LIN {X 0,Y 305.412,Z 307.44,A -85,B 0,C 180,E1 -15880.589,E2 -15880.589} C_VEL
LIN {X 0,Y 305.423,Z 307.439,A -85,B 0,C 180,E1 -15883.655,E2 -15883.655} C_VEL
LIN {X 0,Y 305.438,Z 307.44,A -85,B 0,C 180,E1 -15887.418,E2 -15887.418} C_VEL
LIN {X 0,Y 305.462,Z 307.437,A -85,B 0,C 180,E1 -15891.594,E2 -15891.594} C_VEL
LIN {X 0,Y 305.463,Z 307.435,A -85,B 0,C 180,E1 -15894.886,E2 -15894.886} C_VEL
LIN {X 0,Y 305.507,Z 307.555,A -85,B 0,C 180,E1 -15897.763,E2 -15897.763} C_VEL
LIN {X 0,Y 308.158,Z 320.105,A -85,B 0,C 180,E1 -15901.383,E2 -15901.383} C_VEL
LIN {X 0,Y 309.521,Z 328.593,A -85,B 0,C 180,E1 -15903.719,E2 -15903.719} C_VEL
LIN {X 0,Y 308.772,Z 334.974,A -85,B 0,C 180,E1 -15905.332,E2 -15905.332} C_VEL
LIN {X 0,Y 312.598,Z 362.726,A -85,B 0,C 180,E1 -15906.277,E2 -15906.277} C_VEL
LIN {X 0,Y 314.573,Z 379.937,A -85,B 0,C 180,E1 -15906.819,E2 -15906.819} C_VEL
LIN {X 0,Y 313.206,Z 444.59,A -85,B 0,C 180,E1 -15908.312,E2 -15908.312} C_VEL
LIN {X 0,Y 312.354,Z 458.417,A -85,B 0,C 180,E1 -15908.899,E2 -15908.899} C_VEL
LIN {X 0,Y 311.373,Z 470.835,A -85,B 0,C 180,E1 -15909.693,E2 -15909.693} C_VEL
LIN {X 0,Y 309.988,Z 483.522,A -85,B 0,C 180,E1 -15910.807,E2 -15910.807} C_VEL
LIN {X 0,Y 308.712,Z 494.84,A -85,B 0,C 180,E1 -15912.1,E2 -15912.1} C_VEL
LIN {X 0,Y 307.441,Z 505.618,A -85,B 0,C 180,E1 -15913.671,E2 -15913.671} C_VEL
LIN {X 0,Y 306.35,Z 515.028,A -85,B 0,C 180,E1 -15915.382,E2 -15915.382} C_VEL
LIN {X 0,Y 305.278,Z 523.823,A -85,B 0,C 180,E1 -15917.366,E2 -15917.366} C_VEL
LIN {X 0,Y 304.494,Z 530.826,A -85,B 0,C 180,E1 -15919.359,E2 -15919.359} C_VEL
LIN {X 0,Y 304.015,Z 536.433,A -85,B 0,C 180,E1 -15921.357,E2 -15921.357} C_VEL
LIN {X 0,Y 303.752,Z 540.824,A -85,B 0,C 180,E1 -15923.356,E2 -15923.356} C_VEL
LIN {X 0,Y 303.695,Z 543.143,A -85,B 0,C 180,E1 -15924.688,E2 -15924.688} C_VEL
LIN {X 0,Y 303.704,Z 545.022,A -85,B 0,C 180,E1 -15926.018,E2 -15926.018} C_VEL
LIN {X 0,Y 303.684,Z 546.422,A -85,B 0,C 180,E1 -15927.346,E2 -15927.346} C_VEL
LIN {X 0,Y 303.71,Z 547.415,A -85,B 0,C 180,E1 -15928.673,E2 -15928.673} C_VEL
LIN {X 0,Y 303.765,Z 548.015,A -85,B 0,C 180,E1 -15929.999,E2 -15929.999} C_VEL
LIN {X 0,Y 303.684,Z 548.212,A -85,B 0,C 180,E1 -15931.325,E2 -15931.325} C_VEL
LIN {X 0,Y 303.656,Z 547.975,A -85,B 0,C 180,E1 -15932.652,E2 -15932.652} C_VEL
LIN {X 0,Y 303.659,Z 547.346,A -85,B 0,C 180,E1 -15933.981,E2 -15933.981} C_VEL
LIN {X 0,Y 303.659,Z 546.063,A -85,B 0,C 180,E1 -15935.61,E2 -15935.61} C_VEL
LIN {X 0,Y 303.947,Z 543.046,A -85,B 0,C 180,E1 -15937.974,E2 -15937.974} C_VEL
LIN {X 0,Y 304.413,Z 539.432,A -85,B 0,C 180,E1 -15939.97,E2 -15939.97} C_VEL
LIN {X 0,Y 305.165,Z 534.729,A -85,B 0,C 180,E1 -15941.962,E2 -15941.962} C_VEL
LIN {X 0,Y 306.652,Z 527.682,A -85,B 0,C 180,E1 -15944.262,E2 -15944.262} C_VEL
LIN {X 0,Y 308.048,Z 520.393,A -85,B 0,C 180,E1 -15946.15,E2 -15946.15} C_VEL
LIN {X 0,Y 309.601,Z 512.33,A -85,B 0,C 180,E1 -15947.845,E2 -15947.845} C_VEL
LIN {X 0,Y 311.414,Z 502.899,A -85,B 0,C 180,E1 -15949.443,E2 -15949.443} C_VEL
LIN {X 0,Y 313.302,Z 492.462,A -85,B 0,C 180,E1 -15950.861,E2 -15950.861} C_VEL
LIN {X 0,Y 315.207,Z 480.88,A -85,B 0,C 180,E1 -15952.101,E2 -15952.101} C_VEL
LIN {X 0,Y 316.925,Z 468.596,A -85,B 0,C 180,E1 -15953.093,E2 -15953.093} C_VEL
LIN {X 0,Y 318.276,Z 455.706,A -85,B 0,C 180,E1 -15953.851,E2 -15953.851} C_VEL
LIN {X 0,Y 319.195,Z 443.251,A -85,B 0,C 180,E1 -15954.339,E2 -15954.339} C_VEL
LIN {X 0,Y 320.912,Z 380.563,A -85,B 0,C 180,E1 -15955.776,E2 -15955.776} C_VEL
LIN {X 0,Y 316.937,Z 356.478,A -85,B 0,C 180,E1 -15956.79,E2 -15956.79} C_VEL
LIN {X 0,Y 313.018,Z 337.758,A -85,B 0,C 180,E1 -15957.693,E2 -15957.693} C_VEL
LIN {X 0,Y 311.649,Z 334.114,A -85,B 0,C 180,E1 -15957.962,E2 -15957.962} C_VEL
LIN {X 0,Y 309.652,Z 324.511,A -85,B 0,C 180,E1 -15960.862,E2 -15960.862} C_VEL
LIN {X 0,Y 307.394,Z 314.899,A -85,B 0,C 180,E1 -15963.933,E2 -15963.933} C_VEL
LIN {X 0,Y 305.469,Z 307.44,A -85,B 0,C 180,E1 -15966.496,E2 -15966.496} C_VEL
LIN {X 0,Y 305.455,Z 307.437,A -85,B 0,C 180,E1 -15970.107,E2 -15970.107} C_VEL
LIN {X 0,Y 305.422,Z 307.44,A -85,B 0,C 180,E1 -15973.654,E2 -15973.654} C_VEL
LIN {X 0,Y 305.452,Z 307.436,A -85,B 0,C 180,E1 -15977.414,E2 -15977.414} C_VEL
LIN {X 0,Y 305.472,Z 307.43,A -85,B 0,C 180,E1 -15981.597,E2 -15981.597} C_VEL
LIN {X 0,Y 305.459,Z 307.429,A -85,B 0,C 180,E1 -15984.886,E2 -15984.886} C_VEL
LIN {X 0,Y 305.445,Z 307.43,A -85,B 0,C 180,E1 -15988.355,E2 -15988.355} C_VEL
LIN {X 0,Y 305.509,Z 307.423,A -85,B 0,C 180,E1 -15991.113,E2 -15991.113} C_VEL
LIN {X 0,Y 305.567,Z 307.42,A -85,B 0,C 180,E1 -15994.088,E2 -15994.088} C_VEL
LIN {X 0,Y 305.522,Z 307.427,A -85,B 0,C 180,E1 -15998.405,E2 -15998.405} C_VEL
LIN {X 0,Y 305.586,Z 307.42,A -85,B 0,C 180,E1 -16001.218,E2 -16001.218} C_VEL
LIN {X 0,Y 305.645,Z 307.412,A -85,B 0,C 180,E1 -16005.349,E2 -16005.349} C_VEL
LIN {X 0,Y 305.635,Z 307.413,A -85,B 0,C 180,E1 -16009.4,E2 -16009.4} C_VEL
LIN {X 0,Y 305.809,Z 307.383,A -85,B 0,C 180,E1 -16012.075,E2 -16012.075} C_VEL
LIN {X 0,Y 305.686,Z 307.408,A -85,B 0,C 180,E1 -16014.724,E2 -16014.724} C_VEL
LIN {X 0,Y 305.954,Z 307.375,A -85,B 0,C 180,E1 -16018.684,E2 -16018.684} C_VEL
LIN {X 0,Y 305.954,Z 307.369,A -85,B 0,C 180,E1 -16021.317,E2 -16021.317} C_VEL
LIN {X 0,Y 305.849,Z 307.384,A -85,B 0,C 180,E1 -16026.598,E2 -16026.598} C_VEL
LIN {X 0,Y 305.732,Z 307.394,A -85,B 0,C 180,E1 -16029.26,E2 -16029.26} C_VEL
LIN {X 0,Y 305.586,Z 307.413,A -85,B 0,C 180,E1 -16033.297,E2 -16033.297} C_VEL
LIN {X 0,Y 305.591,Z 307.417,A -85,B 0,C 180,E1 -16036.021,E2 -16036.021} C_VEL
LIN {X 0,Y 305.573,Z 307.422,A -85,B 0,C 180,E1 -16039.445,E2 -16039.445} C_VEL
LIN {X 0,Y 305.488,Z 307.432,A -85,B 0,C 180,E1 -16043.042,E2 -16043.042} C_VEL
LIN {X 0,Y 305.529,Z 307.424,A -85,B 0,C 180,E1 -16046.222,E2 -16046.222} C_VEL
LIN {X 0,Y 305.486,Z 307.427,A -85,B 0,C 180,E1 -16049.048,E2 -16049.048} C_VEL
LIN {X 0,Y 305.44,Z 307.43,A -85,B 0,C 180,E1 -16051.953,E2 -16051.953} C_VEL
LIN {X 0,Y 305.46,Z 307.43,A -85,B 0,C 180,E1 -16055.114,E2 -16055.114} C_VEL
LIN {X 0,Y 305.433,Z 307.431,A -85,B 0,C 180,E1 -16058.526,E2 -16058.526} C_VEL
LIN {X 0,Y 305.438,Z 307.438,A -85,B 0,C 180,E1 -16061.858,E2 -16061.858} C_VEL
LIN {X 0,Y 305.399,Z 307.441,A -85,B 0,C 180,E1 -16065.512,E2 -16065.512} C_VEL
LIN {X 0,Y 305.411,Z 307.441,A -85,B 0,C 180,E1 -16068.139,E2 -16068.139} C_VEL
LIN {X 0,Y 305.461,Z 307.635,A -85,B 0,C 180,E1 -16071.682,E2 -16071.682} C_VEL
LIN {X 0,Y 306.086,Z 309.918,A -85,B 0,C 180,E1 -16072.456,E2 -16072.456} C_VEL
LIN {X 0,Y 313.915,Z 325.345,A -85,B 0,C 180,E1 -16073.763,E2 -16073.763} C_VEL
LIN {X 0,Y 321.808,Z 343.043,A -85,B 0,C 180,E1 -16075.052,E2 -16075.052} C_VEL
LIN {X 0,Y 321.882,Z 347.906,A -85,B 0,C 180,E1 -16075.182,E2 -16075.182} C_VEL
LIN {X 0,Y 319.74,Z 416.224,A -85,B 0,C 180,E1 -16076.715,E2 -16076.715} C_VEL
LIN {X 0,Y 319.076,Z 429.194,A -85,B 0,C 180,E1 -16077.248,E2 -16077.248} C_VEL
LIN {X 0,Y 317.86,Z 442.361,A -85,B 0,C 180,E1 -16078.045,E2 -16078.045} C_VEL
LIN {X 0,Y 316.322,Z 454.752,A -85,B 0,C 180,E1 -16079.084,E2 -16079.084} C_VEL
LIN {X 0,Y 314.924,Z 465.141,A -85,B 0,C 180,E1 -16080.229,E2 -16080.229} C_VEL
LIN {X 0,Y 313.272,Z 475.048,A -85,B 0,C 180,E1 -16081.577,E2 -16081.577} C_VEL
LIN {X 0,Y 311.518,Z 484.552,A -85,B 0,C 180,E1 -16083.18,E2 -16083.18} C_VEL
LIN {X 0,Y 309.735,Z 493.368,A -85,B 0,C 180,E1 -16085.041,E2 -16085.041} C_VEL
LIN {X 0,Y 307.976,Z 501.365,A -85,B 0,C 180,E1 -16087.175,E2 -16087.175} C_VEL
LIN {X 0,Y 306.664,Z 507.305,A -85,B 0,C 180,E1 -16089.194,E2 -16089.194} C_VEL
LIN {X 0,Y 305.632,Z 511.949,A -85,B 0,C 180,E1 -16091.221,E2 -16091.221} C_VEL
LIN {X 0,Y 305.076,Z 514.383,A -85,B 0,C 180,E1 -16092.575,E2 -16092.575} C_VEL
LIN {X 0,Y 304.652,Z 516.358,A -85,B 0,C 180,E1 -16093.93,E2 -16093.93} C_VEL
LIN {X 0,Y 304.191,Z 518.541,A -85,B 0,C 180,E1 -16096.019,E2 -16096.019} C_VEL
LIN {X 0,Y 303.846,Z 519.689,A -85,B 0,C 180,E1 -16097.986,E2 -16097.986} C_VEL
LIN {X 0,Y 303.634,Z 519.884,A -85,B 0,C 180,E1 -16100.676,E2 -16100.676} C_VEL
LIN {X 0,Y 303.703,Z 519.354,A -85,B 0,C 180,E1 -16102.02,E2 -16102.02} C_VEL
LIN {X 0,Y 303.857,Z 517.831,A -85,B 0,C 180,E1 -16104.027,E2 -16104.027} C_VEL
LIN {X 0,Y 304.029,Z 514.328,A -85,B 0,C 180,E1 -16106.688,E2 -16106.688} C_VEL
LIN {X 0,Y 304.459,Z 510.533,A -85,B 0,C 180,E1 -16108.678,E2 -16108.678} C_VEL
LIN {X 0,Y 304.937,Z 505.635,A -85,B 0,C 180,E1 -16110.661,E2 -16110.661} C_VEL
LIN {X 0,Y 305.759,Z 499.464,A -85,B 0,C 180,E1 -16112.636,E2 -16112.636} C_VEL
LIN {X 0,Y 306.778,Z 491.775,A -85,B 0,C 180,E1 -16114.6,E2 -16114.6} C_VEL
LIN {X 0,Y 307.98,Z 482.158,A -85,B 0,C 180,E1 -16116.552,E2 -16116.552} C_VEL
LIN {X 0,Y 309.261,Z 472.211,A -85,B 0,C 180,E1 -16118.166,E2 -16118.166} C_VEL
LIN {X 0,Y 310.521,Z 460.956,A -85,B 0,C 180,E1 -16119.609,E2 -16119.609} C_VEL
LIN {X 0,Y 311.568,Z 449.946,A -85,B 0,C 180,E1 -16120.726,E2 -16120.726} C_VEL
LIN {X 0,Y 312.416,Z 437.754,A -85,B 0,C 180,E1 -16121.682,E2 -16121.682} C_VEL
LIN {X 0,Y 313.208,Z 424.771,A -85,B 0,C 180,E1 -16122.391,E2 -16122.391} C_VEL
LIN {X 0,Y 313.644,Z 410.959,A -85,B 0,C 180,E1 -16122.867,E2 -16122.867} C_VEL
LIN {X 0,Y 315.279,Z 336.381,A -85,B 0,C 180,E1 -16124.543,E2 -16124.543} C_VEL
LIN {X 0,Y 313.144,Z 328.581,A -85,B 0,C 180,E1 -16124.877,E2 -16124.877} C_VEL
LIN {X 0,Y 305.913,Z 308.922,A -85,B 0,C 180,E1 -16125.893,E2 -16125.893} C_VEL
LIN {X 0,Y 305.603,Z 307.419,A -85,B 0,C 180,E1 -16126.363,E2 -16126.363} C_VEL
LIN {X 0,Y 305.5,Z 307.429,A -85,B 0,C 180,E1 -16130.187,E2 -16130.187} C_VEL
LIN {X 0,Y 305.479,Z 307.43,A -85,B 0,C 180,E1 -16134.465,E2 -16134.465} C_VEL
LIN {X 0,Y 305.459,Z 307.433,A -85,B 0,C 180,E1 -16137.398,E2 -16137.398} C_VEL
LIN {X 0,Y 305.435,Z 307.436,A -85,B 0,C 180,E1 -16140.413,E2 -16140.413} C_VEL
LIN {X 0,Y 305.47,Z 307.431,A -85,B 0,C 180,E1 -16144.079,E2 -16144.079} C_VEL
LIN {X 0,Y 305.459,Z 307.435,A -85,B 0,C 180,E1 -16146.743,E2 -16146.743} C_VEL
LIN {X 0,Y 305.414,Z 307.437,A -85,B 0,C 180,E1 -16150.59,E2 -16150.59} C_VEL
LIN {X 0,Y 305.425,Z 307.439,A -85,B 0,C 180,E1 -16153.656,E2 -16153.656} C_VEL
LIN {X 0,Y 305.44,Z 307.435,A -85,B 0,C 180,E1 -16157.418,E2 -16157.418} C_VEL
LIN {X 0,Y 305.404,Z 307.436,A -85,B 0,C 180,E1 -16158.391,E2 -16158.391} C_VEL
LIN {X 0,Y 304.724,Z 307.528,A -85,B 0,C 180,E1 -16159.492,E2 -16159.492} C_VEL
LIN {X 0,Y 301.902,Z 307.879,A -85,B 0,C 180,E1 -16161.287,E2 -16161.287} C_VEL
LIN {X 0,Y 299.516,Z 308.174,A -85,B 0,C 180,E1 -16162.742,E2 -16162.742} C_VEL
LIN {X 0,Y 298.485,Z 308.3,A -85,B 0,C 180,E1 -16163.868,E2 -16163.868} C_VEL
LIN {X 0,Y 298.395,Z 308.308,A -85,B 0,C 180,E1 -16164.25,E2 -16164.25} C_VEL
LIN {X 0,Y 298.393,Z 308.314,A -85,B 0,C 180,E1 -16167.986,E2 -16167.986} C_VEL
LIN {X 0,Y 298.416,Z 308.311,A -85,B 0,C 180,E1 -16171.899,E2 -16171.899} C_VEL
LIN {X 0,Y 298.429,Z 308.3,A -85,B 0,C 180,E1 -16174.918,E2 -16174.918} C_VEL
LIN {X 0,Y 298.407,Z 308.315,A -85,B 0,C 180,E1 -16177.862,E2 -16177.862} C_VEL
LIN {X 0,Y 298.508,Z 308.298,A -85,B 0,C 180,E1 -16180.754,E2 -16180.754} C_VEL
LIN {X 0,Y 298.591,Z 308.28,A -85,B 0,C 180,E1 -16184.994,E2 -16184.994} C_VEL
LIN {X 0,Y 298.587,Z 308.288,A -85,B 0,C 180,E1 -16189.146,E2 -16189.146} C_VEL
LIN {X 0,Y 298.703,Z 308.277,A -85,B 0,C 180,E1 -16191.884,E2 -16191.884} C_VEL
LIN {X 0,Y 298.632,Z 308.276,A -85,B 0,C 180,E1 -16194.598,E2 -16194.598} C_VEL
LIN {X 0,Y 298.907,Z 308.25,A -85,B 0,C 180,E1 -16198.652,E2 -16198.652} C_VEL
LIN {X 0,Y 298.914,Z 308.248,A -85,B 0,C 180,E1 -16201.347,E2 -16201.347} C_VEL
LIN {X 0,Y 298.737,Z 308.267,A -85,B 0,C 180,E1 -16206.755,E2 -16206.755} C_VEL
LIN {X 0,Y 298.629,Z 308.282,A -85,B 0,C 180,E1 -16209.482,E2 -16209.482} C_VEL
LIN {X 0,Y 298.548,Z 308.292,A -85,B 0,C 180,E1 -16213.615,E2 -16213.615} C_VEL
LIN {X 0,Y 298.488,Z 308.305,A -85,B 0,C 180,E1 -16216.412,E2 -16216.412} C_VEL
LIN {X 0,Y 298.449,Z 308.306,A -85,B 0,C 180,E1 -16219.618,E2 -16219.618} C_VEL
LIN {X 0,Y 298.424,Z 308.309,A -85,B 0,C 180,E1 -16223.6,E2 -16223.6} C_VEL
LIN {X 0,Y 298.41,Z 308.314,A -85,B 0,C 180,E1 -16226.582,E2 -16226.582} C_VEL
LIN {X 0,Y 298.364,Z 308.318,A -85,B 0,C 180,E1 -16229.647,E2 -16229.647} C_VEL
LIN {X 0,Y 298.396,Z 308.317,A -85,B 0,C 180,E1 -16232.8,E2 -16232.8} C_VEL
LIN {X 0,Y 298.43,Z 308.312,A -85,B 0,C 180,E1 -16236.802,E2 -16236.802} C_VEL
LIN {X 0,Y 298.376,Z 308.318,A -85,B 0,C 180,E1 -16239.491,E2 -16239.491} C_VEL
LIN {X 0,Y 298.373,Z 308.32,A -85,B 0,C 180,E1 -16243.097,E2 -16243.097} C_VEL
LIN {X 0,Y 298.373,Z 308.317,A -85,B 0,C 180,E1 -16246.914,E2 -16246.914} C_VEL
LIN {X 0,Y 298.387,Z 308.316,A -85,B 0,C 180,E1 -16251.01,E2 -16251.01} C_VEL
LIN {X 0,Y 298.418,Z 308.314,A -85,B 0,C 180,E1 -16253.929,E2 -16253.929} C_VEL
LIN {X 0,Y 298.478,Z 308.417,A -85,B 0,C 180,E1 -16257.366,E2 -16257.366} C_VEL
LIN {X 0,Y 301.069,Z 320.78,A -85,B 0,C 180,E1 -16261.028,E2 -16261.028} C_VEL
LIN {X 0,Y 302.543,Z 329.288,A -85,B 0,C 180,E1 -16263.437,E2 -16263.437} C_VEL
LIN {X 0,Y 301.955,Z 334.637,A -85,B 0,C 180,E1 -16264.826,E2 -16264.826} C_VEL
LIN {X 0,Y 305.753,Z 362.062,A -85,B 0,C 180,E1 -16265.792,E2 -16265.792} C_VEL
LIN {X 0,Y 307.897,Z 380.351,A -85,B 0,C 180,E1 -16266.388,E2 -16266.388} C_VEL
LIN {X 0,Y 306.579,Z 443.282,A -85,B 0,C 180,E1 -16267.863,E2 -16267.863} C_VEL
LIN {X 0,Y 305.743,Z 456.666,A -85,B 0,C 180,E1 -16268.42,E2 -16268.42} C_VEL
LIN {X 0,Y 304.699,Z 469.491,A -85,B 0,C 180,E1 -16269.228,E2 -16269.228} C_VEL
LIN {X 0,Y 303.478,Z 480.858,A -85,B 0,C 180,E1 -16270.202,E2 -16270.202} C_VEL
LIN {X 0,Y 302.022,Z 492.589,A -85,B 0,C 180,E1 -16271.514,E2 -16271.514} C_VEL
LIN {X 0,Y 300.825,Z 503.17,A -85,B 0,C 180,E1 -16273.02,E2 -16273.02} C_VEL
LIN {X 0,Y 299.703,Z 512.814,A -85,B 0,C 180,E1 -16274.733,E2 -16274.733} C_VEL
LIN {X 0,Y 298.472,Z 521.816,A -85,B 0,C 180,E1 -16276.727,E2 -16276.727} C_VEL
LIN {X 0,Y 297.546,Z 529.18,A -85,B 0,C 180,E1 -16278.762,E2 -16278.762} C_VEL
LIN {X 0,Y 297.093,Z 534.164,A -85,B 0,C 180,E1 -16280.468,E2 -16280.468} C_VEL
LIN {X 0,Y 296.777,Z 538.998,A -85,B 0,C 180,E1 -16282.515,E2 -16282.515} C_VEL
LIN {X 0,Y 296.62,Z 542.689,A -85,B 0,C 180,E1 -16284.561,E2 -16284.561} C_VEL
LIN {X 0,Y 296.616,Z 544.593,A -85,B 0,C 180,E1 -16285.923,E2 -16285.923} C_VEL
LIN {X 0,Y 296.607,Z 546.027,A -85,B 0,C 180,E1 -16287.283,E2 -16287.283} C_VEL
LIN {X 0,Y 296.622,Z 547.038,A -85,B 0,C 180,E1 -16288.641,E2 -16288.641} C_VEL
LIN {X 0,Y 296.673,Z 547.656,A -85,B 0,C 180,E1 -16289.999,E2 -16289.999} C_VEL
LIN {X 0,Y 296.596,Z 547.877,A -85,B 0,C 180,E1 -16291.357,E2 -16291.357} C_VEL
LIN {X 0,Y 296.579,Z 547.673,A -85,B 0,C 180,E1 -16292.716,E2 -16292.716} C_VEL
LIN {X 0,Y 296.572,Z 547.061,A -85,B 0,C 180,E1 -16294.076,E2 -16294.076} C_VEL
LIN {X 0,Y 296.587,Z 545.932,A -85,B 0,C 180,E1 -16295.591,E2 -16295.591} C_VEL
LIN {X 0,Y 296.887,Z 542.837,A -85,B 0,C 180,E1 -16298.165,E2 -16298.165} C_VEL
LIN {X 0,Y 297.398,Z 539.265,A -85,B 0,C 180,E1 -16300.208,E2 -16300.208} C_VEL
LIN {X 0,Y 298.183,Z 534.607,A -85,B 0,C 180,E1 -16302.246,E2 -16302.246} C_VEL
LIN {X 0,Y 299.769,Z 527.608,A -85,B 0,C 180,E1 -16304.597,E2 -16304.597} C_VEL
LIN {X 0,Y 301.357,Z 519.808,A -85,B 0,C 180,E1 -16306.664,E2 -16306.664} C_VEL
LIN {X 0,Y 303.168,Z 510.646,A -85,B 0,C 180,E1 -16308.586,E2 -16308.586} C_VEL
LIN {X 0,Y 305.175,Z 500.933,A -85,B 0,C 180,E1 -16310.208,E2 -16310.208} C_VEL
LIN {X 0,Y 307.202,Z 490.161,A -85,B 0,C 180,E1 -16311.647,E2 -16311.647} C_VEL
LIN {X 0,Y 308.945,Z 479.683,A -85,B 0,C 180,E1 -16312.75,E2 -16312.75} C_VEL
LIN {X 0,Y 310.577,Z 468.216,A -85,B 0,C 180,E1 -16313.681,E2 -16313.681} C_VEL
LIN {X 0,Y 311.967,Z 455.318,A -85,B 0,C 180,E1 -16314.452,E2 -16314.452} C_VEL
LIN {X 0,Y 312.933,Z 442.835,A -85,B 0,C 180,E1 -16314.947,E2 -16314.947} C_VEL
LIN {X 0,Y 314.672,Z 381.223,A -85,B 0,C 180,E1 -16316.387,E2 -16316.387} C_VEL
LIN {X 0,Y 310.614,Z 356.75,A -85,B 0,C 180,E1 -16317.455,E2 -16317.455} C_VEL
LIN {X 0,Y 306.958,Z 339.936,A -85,B 0,C 180,E1 -16318.311,E2 -16318.311} C_VEL
LIN {X 0,Y 304.432,Z 333.652,A -85,B 0,C 180,E1 -16318.813,E2 -16318.813} C_VEL
LIN {X 0,Y 301.993,Z 322.401,A -85,B 0,C 180,E1 -16322.36,E2 -16322.36} C_VEL
LIN {X 0,Y 299.372,Z 311.813,A -85,B 0,C 180,E1 -16325.936,E2 -16325.936} C_VEL
LIN {X 0,Y 298.41,Z 308.314,A -85,B 0,C 180,E1 -16327.223,E2 -16327.223} C_VEL
LIN {X 0,Y 298.381,Z 308.314,A -85,B 0,C 180,E1 -16331.261,E2 -16331.261} C_VEL
LIN {X 0,Y 298.351,Z 308.322,A -85,B 0,C 180,E1 -16335.034,E2 -16335.034} C_VEL
LIN {X 0,Y 298.381,Z 308.313,A -85,B 0,C 180,E1 -16338.738,E2 -16338.738} C_VEL
LIN {X 0,Y 298.41,Z 308.308,A -85,B 0,C 180,E1 -16342.241,E2 -16342.241} C_VEL
LIN {X 0,Y 298.404,Z 308.307,A -85,B 0,C 180,E1 -16345.581,E2 -16345.581} C_VEL
LIN {X 0,Y 298.388,Z 308.309,A -85,B 0,C 180,E1 -16348.79,E2 -16348.79} C_VEL
LIN {X 0,Y 298.455,Z 308.299,A -85,B 0,C 180,E1 -16351.904,E2 -16351.904} C_VEL
LIN {X 0,Y 298.482,Z 308.298,A -85,B 0,C 180,E1 -16354.924,E2 -16354.924} C_VEL
LIN {X 0,Y 298.454,Z 308.298,A -85,B 0,C 180,E1 -16359.316,E2 -16359.316} C_VEL
LIN {X 0,Y 298.534,Z 308.298,A -85,B 0,C 180,E1 -16362.179,E2 -16362.179} C_VEL
LIN {X 0,Y 298.59,Z 308.291,A -85,B 0,C 180,E1 -16364.995,E2 -16364.995} C_VEL
LIN {X 0,Y 298.59,Z 308.291,A -85,B 0,C 180,E1 -16369.147,E2 -16369.147} C_VEL
LIN {X 0,Y 298.755,Z 308.262,A -85,B 0,C 180,E1 -16371.886,E2 -16371.886} C_VEL
LIN {X 0,Y 298.657,Z 308.284,A -85,B 0,C 180,E1 -16374.599,E2 -16374.599} C_VEL
LIN {X 0,Y 298.92,Z 308.251,A -85,B 0,C 180,E1 -16378.653,E2 -16378.653} C_VEL
LIN {X 0,Y 298.92,Z 308.245,A -85,B 0,C 180,E1 -16381.348,E2 -16381.348} C_VEL
LIN {X 0,Y 298.795,Z 308.264,A -85,B 0,C 180,E1 -16386.754,E2 -16386.754} C_VEL
LIN {X 0,Y 298.677,Z 308.273,A -85,B 0,C 180,E1 -16389.481,E2 -16389.481} C_VEL
LIN {X 0,Y 298.549,Z 308.289,A -85,B 0,C 180,E1 -16393.616,E2 -16393.616} C_VEL
LIN {X 0,Y 298.546,Z 308.295,A -85,B 0,C 180,E1 -16396.409,E2 -16396.409} C_VEL
LIN {X 0,Y 298.508,Z 308.301,A -85,B 0,C 180,E1 -16399.655,E2 -16399.655} C_VEL
LIN {X 0,Y 298.455,Z 308.308,A -85,B 0,C 180,E1 -16403.598,E2 -16403.598} C_VEL
LIN {X 0,Y 298.484,Z 308.302,A -85,B 0,C 180,E1 -16406.575,E2 -16406.575} C_VEL
LIN {X 0,Y 298.414,Z 308.31,A -85,B 0,C 180,E1 -16409.642,E2 -16409.642} C_VEL
LIN {X 0,Y 298.393,Z 308.308,A -85,B 0,C 180,E1 -16412.801,E2 -16412.801} C_VEL
LIN {X 0,Y 298.44,Z 308.308,A -85,B 0,C 180,E1 -16416.807,E2 -16416.807} C_VEL
LIN {X 0,Y 298.384,Z 308.312,A -85,B 0,C 180,E1 -16421.088,E2 -16421.088} C_VEL
LIN {X 0,Y 298.398,Z 308.313,A -85,B 0,C 180,E1 -16423.104,E2 -16423.104} C_VEL
LIN {X 0,Y 298.37,Z 308.321,A -85,B 0,C 180,E1 -16426.916,E2 -16426.916} C_VEL
LIN {X 0,Y 298.362,Z 308.328,A -85,B 0,C 180,E1 -16430.899,E2 -16430.899} C_VEL
LIN {X 0,Y 298.905,Z 310.268,A -85,B 0,C 180,E1 -16431.587,E2 -16431.587} C_VEL
LIN {X 0,Y 300.751,Z 313.796,A -85,B 0,C 180,E1 -16431.916,E2 -16431.916} C_VEL
LIN {X 0,Y 308.446,Z 328.838,A -85,B 0,C 180,E1 -16433.244,E2 -16433.244} C_VEL
LIN {X 0,Y 315.724,Z 345.313,A -85,B 0,C 180,E1 -16434.478,E2 -16434.478} C_VEL
LIN {X 0,Y 313.433,Z 417.477,A -85,B 0,C 180,E1 -16436.142,E2 -16436.142} C_VEL
LIN {X 0,Y 312.713,Z 430.572,A -85,B 0,C 180,E1 -16436.71,E2 -16436.71} C_VEL
LIN {X 0,Y 311.474,Z 443.2,A -85,B 0,C 180,E1 -16437.501,E2 -16437.501} C_VEL
LIN {X 0,Y 309.881,Z 455.439,A -85,B 0,C 180,E1 -16438.559,E2 -16438.559} C_VEL
LIN {X 0,Y 308.405,Z 465.76,A -85,B 0,C 180,E1 -16439.723,E2 -16439.723} C_VEL
LIN {X 0,Y 306.527,Z 476.414,A -85,B 0,C 180,E1 -16441.219,E2 -16441.219} C_VEL
LIN {X 0,Y 304.694,Z 485.937,A -85,B 0,C 180,E1 -16442.901,E2 -16442.901} C_VEL
LIN {X 0,Y 302.801,Z 494.732,A -85,B 0,C 180,E1 -16444.85,E2 -16444.85} C_VEL
LIN {X 0,Y 301.019,Z 502.377,A -85,B 0,C 180,E1 -16446.98,E2 -16446.98} C_VEL
LIN {X 0,Y 299.867,Z 507.273,A -85,B 0,C 180,E1 -16448.7,E2 -16448.7} C_VEL
LIN {X 0,Y 298.743,Z 511.997,A -85,B 0,C 180,E1 -16450.771,E2 -16450.771} C_VEL
LIN {X 0,Y 297.916,Z 515.569,A -85,B 0,C 180,E1 -16452.85,E2 -16452.85} C_VEL
LIN {X 0,Y 297.319,Z 518.097,A -85,B 0,C 180,E1 -16454.93,E2 -16454.93} C_VEL
LIN {X 0,Y 297.052,Z 519.26,A -85,B 0,C 180,E1 -16456.315,E2 -16456.315} C_VEL
LIN {X 0,Y 296.802,Z 519.974,A -85,B 0,C 180,E1 -16457.696,E2 -16457.696} C_VEL
LIN {X 0,Y 296.54,Z 520.234,A -85,B 0,C 180,E1 -16460.451,E2 -16460.451} C_VEL
LIN {X 0,Y 296.606,Z 519.766,A -85,B 0,C 180,E1 -16461.828,E2 -16461.828} C_VEL
LIN {X 0,Y 296.765,Z 518.102,A -85,B 0,C 180,E1 -16464.076,E2 -16464.076} C_VEL
LIN {X 0,Y 296.937,Z 514.87,A -85,B 0,C 180,E1 -16466.609,E2 -16466.609} C_VEL
LIN {X 0,Y 297.379,Z 511.144,A -85,B 0,C 180,E1 -16468.647,E2 -16468.647} C_VEL
LIN {X 0,Y 297.858,Z 506.322,A -85,B 0,C 180,E1 -16470.677,E2 -16470.677} C_VEL
LIN {X 0,Y 298.685,Z 500.235,A -85,B 0,C 180,E1 -16472.698,E2 -16472.698} C_VEL
LIN {X 0,Y 299.731,Z 492.678,A -85,B 0,C 180,E1 -16474.708,E2 -16474.708} C_VEL
LIN {X 0,Y 300.747,Z 484.954,A -85,B 0,C 180,E1 -16476.374,E2 -16476.374} C_VEL
LIN {X 0,Y 302.138,Z 474.455,A -85,B 0,C 180,E1 -16478.192,E2 -16478.192} C_VEL
LIN {X 0,Y 303.422,Z 463.775,A -85,B 0,C 180,E1 -16479.668,E2 -16479.668} C_VEL
LIN {X 0,Y 304.527,Z 453.401,A -85,B 0,C 180,E1 -16480.808,E2 -16480.808} C_VEL
LIN {X 0,Y 305.47,Z 440.987,A -85,B 0,C 180,E1 -16481.867,E2 -16481.867} C_VEL
LIN {X 0,Y 306.371,Z 427.838,A -85,B 0,C 180,E1 -16482.672,E2 -16482.672} C_VEL
LIN {X 0,Y 306.864,Z 414.521,A -85,B 0,C 180,E1 -16483.198,E2 -16483.198} C_VEL
LIN {X 0,Y 308.72,Z 337.899,A -85,B 0,C 180,E1 -16484.961,E2 -16484.961} C_VEL
LIN {X 0,Y 306.496,Z 330.201,A -85,B 0,C 180,E1 -16485.31,E2 -16485.31} C_VEL
LIN {X 0,Y 299.55,Z 311.529,A -85,B 0,C 180,E1 -16486.301,E2 -16486.301} C_VEL
LIN {X 0,Y 298.745,Z 309.24,A -85,B 0,C 180,E1 -16486.442,E2 -16486.442} C_VEL
LIN {X 0,Y 298.534,Z 308.3,A -85,B 0,C 180,E1 -16486.762,E2 -16486.762} C_VEL
LIN {X 0,Y 298.488,Z 308.302,A -85,B 0,C 180,E1 -16489.64,E2 -16489.64} C_VEL
LIN {X 0,Y 298.425,Z 308.307,A -85,B 0,C 180,E1 -16493.601,E2 -16493.601} C_VEL
LIN {X 0,Y 298.412,Z 308.31,A -85,B 0,C 180,E1 -16496.583,E2 -16496.583} C_VEL
LIN {X 0,Y 298.398,Z 308.312,A -85,B 0,C 180,E1 -16499.644,E2 -16499.644} C_VEL
LIN {X 0,Y 298.398,Z 308.316,A -85,B 0,C 180,E1 -16502.801,E2 -16502.801} C_VEL
LIN {X 0,Y 298.433,Z 308.311,A -85,B 0,C 180,E1 -16506.803,E2 -16506.803} C_VEL
LIN {X 0,Y 298.379,Z 308.315,A -85,B 0,C 180,E1 -16509.492,E2 -16509.492} C_VEL
LIN {X 0,Y 298.375,Z 308.317,A -85,B 0,C 180,E1 -16513.097,E2 -16513.097} C_VEL
LIN {X 0,Y 298.376,Z 308.314,A -85,B 0,C 180,E1 -16516.915,E2 -16516.915} C_VEL
LIN {X 0,Y 298.359,Z 308.318,A -85,B 0,C 180,E1 -16521.018,E2 -16521.018} C_VEL
LIN {X 0,Y 298.395,Z 308.308,A -85,B 0,C 180,E1 -16524.25,E2 -16524.25} C_VEL
LIN {X 0,Y 297.698,Z 308.397,A -85,B 0,C 180,E1 -16525.377,E2 -16525.377} C_VEL
LIN {X 0,Y 294.797,Z 308.759,A -85,B 0,C 180,E1 -16527.211,E2 -16527.211} C_VEL
LIN {X 0,Y 292.389,Z 309.062,A -85,B 0,C 180,E1 -16528.7,E2 -16528.7} C_VEL
LIN {X 0,Y 291.416,Z 309.185,A -85,B 0,C 180,E1 -16529.854,E2 -16529.854} C_VEL
LIN {X 0,Y 291.368,Z 309.189,A -85,B 0,C 180,E1 -16530.245,E2 -16530.245} C_VEL
LIN {X 0,Y 291.353,Z 309.182,A -85,B 0,C 180,E1 -16534.265,E2 -16534.265} C_VEL
LIN {X 0,Y 291.364,Z 309.187,A -85,B 0,C 180,E1 -16537.298,E2 -16537.298} C_VEL
LIN {X 0,Y 291.445,Z 309.18,A -85,B 0,C 180,E1 -16540.269,E2 -16540.269} C_VEL
LIN {X 0,Y 291.503,Z 309.162,A -85,B 0,C 180,E1 -16544.665,E2 -16544.665} C_VEL
LIN {X 0,Y 291.533,Z 309.167,A -85,B 0,C 180,E1 -16548.88,E2 -16548.88} C_VEL
LIN {X 0,Y 291.656,Z 309.153,A -85,B 0,C 180,E1 -16551.687,E2 -16551.687} C_VEL
LIN {X 0,Y 291.602,Z 309.152,A -85,B 0,C 180,E1 -16554.467,E2 -16554.467} C_VEL
LIN {X 0,Y 291.875,Z 309.126,A -85,B 0,C 180,E1 -16558.62,E2 -16558.62} C_VEL
LIN {X 0,Y 291.88,Z 309.124,A -85,B 0,C 180,E1 -16561.379,E2 -16561.379} C_VEL
LIN {X 0,Y 291.69,Z 309.143,A -85,B 0,C 180,E1 -16566.919,E2 -16566.919} C_VEL
LIN {X 0,Y 291.572,Z 309.161,A -85,B 0,C 180,E1 -16569.714,E2 -16569.714} C_VEL
LIN {X 0,Y 291.519,Z 309.168,A -85,B 0,C 180,E1 -16573.95,E2 -16573.95} C_VEL
LIN {X 0,Y 291.432,Z 309.183,A -85,B 0,C 180,E1 -16576.821,E2 -16576.821} C_VEL
LIN {X 0,Y 291.395,Z 309.185,A -85,B 0,C 180,E1 -16579.841,E2 -16579.841} C_VEL
LIN {X 0,Y 291.363,Z 309.19,A -85,B 0,C 180,E1 -16584.208,E2 -16584.208} C_VEL
LIN {X 0,Y 291.354,Z 309.192,A -85,B 0,C 180,E1 -16587.278,E2 -16587.278} C_VEL
LIN {X 0,Y 291.307,Z 309.198,A -85,B 0,C 180,E1 -16590.44,E2 -16590.44} C_VEL
LIN {X 0,Y 291.346,Z 309.192,A -85,B 0,C 180,E1 -16593.698,E2 -16593.698} C_VEL
LIN {X 0,Y 291.361,Z 309.194,A -85,B 0,C 180,E1 -16597.249,E2 -16597.249} C_VEL
LIN {X 0,Y 291.303,Z 309.198,A -85,B 0,C 180,E1 -16600.647,E2 -16600.647} C_VEL
LIN {X 0,Y 291.284,Z 309.199,A -85,B 0,C 180,E1 -16604.403,E2 -16604.403} C_VEL
LIN {X 0,Y 291.297,Z 309.197,A -85,B 0,C 180,E1 -16608.411,E2 -16608.411} C_VEL
LIN {X 0,Y 291.337,Z 309.196,A -85,B 0,C 180,E1 -16611.155,E2 -16611.155} C_VEL
LIN {X 0,Y 291.362,Z 309.192,A -85,B 0,C 180,E1 -16614.625,E2 -16614.625} C_VEL
LIN {X 0,Y 291.409,Z 309.396,A -85,B 0,C 180,E1 -16616.981,E2 -16616.981} C_VEL
LIN {X 0,Y 293.711,Z 320.009,A -85,B 0,C 180,E1 -16620.23,E2 -16620.23} C_VEL
LIN {X 0,Y 295.507,Z 329.966,A -85,B 0,C 180,E1 -16623.135,E2 -16623.135} C_VEL
LIN {X 0,Y 295.188,Z 334.296,A -85,B 0,C 180,E1 -16624.299,E2 -16624.299} C_VEL
LIN {X 0,Y 299.234,Z 363.733,A -85,B 0,C 180,E1 -16625.367,E2 -16625.367} C_VEL
LIN {X 0,Y 301.219,Z 381.077,A -85,B 0,C 180,E1 -16625.945,E2 -16625.945} C_VEL
LIN {X 0,Y 299.869,Z 443.076,A -85,B 0,C 180,E1 -16627.431,E2 -16627.431} C_VEL
LIN {X 0,Y 299,Z 456.417,A -85,B 0,C 180,E1 -16627.999,E2 -16627.999} C_VEL
LIN {X 0,Y 297.934,Z 469.226,A -85,B 0,C 180,E1 -16628.825,E2 -16628.825} C_VEL
LIN {X 0,Y 296.563,Z 481.373,A -85,B 0,C 180,E1 -16629.901,E2 -16629.901} C_VEL
LIN {X 0,Y 295.081,Z 492.952,A -85,B 0,C 180,E1 -16631.243,E2 -16631.243} C_VEL
LIN {X 0,Y 293.853,Z 503.412,A -85,B 0,C 180,E1 -16632.783,E2 -16632.783} C_VEL
LIN {X 0,Y 292.777,Z 512.293,A -85,B 0,C 180,E1 -16634.404,E2 -16634.404} C_VEL
LIN {X 0,Y 291.534,Z 521.168,A -85,B 0,C 180,E1 -16636.405,E2 -16636.405} C_VEL
LIN {X 0,Y 290.522,Z 528.584,A -85,B 0,C 180,E1 -16638.487,E2 -16638.487} C_VEL
LIN {X 0,Y 290.058,Z 533.621,A -85,B 0,C 180,E1 -16640.234,E2 -16640.234} C_VEL
LIN {X 0,Y 289.705,Z 538.499,A -85,B 0,C 180,E1 -16642.332,E2 -16642.332} C_VEL
LIN {X 0,Y 289.556,Z 542.235,A -85,B 0,C 180,E1 -16644.428,E2 -16644.428} C_VEL
LIN {X 0,Y 289.533,Z 544.159,A -85,B 0,C 180,E1 -16645.823,E2 -16645.823} C_VEL
LIN {X 0,Y 289.532,Z 545.632,A -85,B 0,C 180,E1 -16647.216,E2 -16647.216} C_VEL
LIN {X 0,Y 289.536,Z 546.662,A -85,B 0,C 180,E1 -16648.608,E2 -16648.608} C_VEL
LIN {X 0,Y 289.583,Z 547.298,A -85,B 0,C 180,E1 -16649.999,E2 -16649.999} C_VEL
LIN {X 0,Y 289.512,Z 547.537,A -85,B 0,C 180,E1 -16651.39,E2 -16651.39} C_VEL
LIN {X 0,Y 289.504,Z 547.37,A -85,B 0,C 180,E1 -16652.782,E2 -16652.782} C_VEL
LIN {X 0,Y 289.48,Z 545.856,A -85,B 0,C 180,E1 -16655.498,E2 -16655.498} C_VEL
LIN {X 0,Y 289.581,Z 544.422,A -85,B 0,C 180,E1 -16656.969,E2 -16656.969} C_VEL
LIN {X 0,Y 290.005,Z 541.546,A -85,B 0,C 180,E1 -16659.062,E2 -16659.062} C_VEL
LIN {X 0,Y 290.642,Z 537.659,A -85,B 0,C 180,E1 -16661.153,E2 -16661.153} C_VEL
LIN {X 0,Y 291.635,Z 532.667,A -85,B 0,C 180,E1 -16663.234,E2 -16663.234} C_VEL
LIN {X 0,Y 293.128,Z 526.421,A -85,B 0,C 180,E1 -16665.291,E2 -16665.291} C_VEL
LIN {X 0,Y 294.806,Z 518.627,A -85,B 0,C 180,E1 -16667.342,E2 -16667.342} C_VEL
LIN {X 0,Y 296.458,Z 510.742,A -85,B 0,C 180,E1 -16669.023,E2 -16669.023} C_VEL
LIN {X 0,Y 298.519,Z 501.116,A -85,B 0,C 180,E1 -16670.679,E2 -16670.679} C_VEL
LIN {X 0,Y 300.632,Z 490.452,A -85,B 0,C 180,E1 -16672.145,E2 -16672.145} C_VEL
LIN {X 0,Y 302.436,Z 480.149,A -85,B 0,C 180,E1 -16673.268,E2 -16673.268} C_VEL
LIN {X 0,Y 304.27,Z 467.844,A -85,B 0,C 180,E1 -16674.294,E2 -16674.294} C_VEL
LIN {X 0,Y 305.717,Z 454.932,A -85,B 0,C 180,E1 -16675.077,E2 -16675.077} C_VEL
LIN {X 0,Y 306.71,Z 442.421,A -85,B 0,C 180,E1 -16675.58,E2 -16675.58} C_VEL
LIN {X 0,Y 308.536,Z 382.541,A -85,B 0,C 180,E1 -16676.998,E2 -16676.998} C_VEL
LIN {X 0,Y 304.787,Z 359.56,A -85,B 0,C 180,E1 -16678.028,E2 -16678.028} C_VEL
LIN {X 0,Y 301.379,Z 343.152,A -85,B 0,C 180,E1 -16678.874,E2 -16678.874} C_VEL
LIN {X 0,Y 297.207,Z 333.325,A -85,B 0,C 180,E1 -16679.676,E2 -16679.676} C_VEL
LIN {X 0,Y 294.65,Z 321.968,A -85,B 0,C 180,E1 -16683.403,E2 -16683.403} C_VEL
LIN {X 0,Y 292.54,Z 313.464,A -85,B 0,C 180,E1 -16686.38,E2 -16686.38} C_VEL
LIN {X 0,Y 291.361,Z 309.193,A -85,B 0,C 180,E1 -16687.983,E2 -16687.983} C_VEL
LIN {X 0,Y 291.323,Z 309.193,A -85,B 0,C 180,E1 -16691.595,E2 -16691.595} C_VEL
LIN {X 0,Y 291.287,Z 309.2,A -85,B 0,C 180,E1 -16695.598,E2 -16695.598} C_VEL
LIN {X 0,Y 291.329,Z 309.19,A -85,B 0,C 180,E1 -16699.357,E2 -16699.357} C_VEL
LIN {X 0,Y 291.404,Z 309.184,A -85,B 0,C 180,E1 -16702.919,E2 -16702.919} C_VEL
LIN {X 0,Y 291.341,Z 309.19,A -85,B 0,C 180,E1 -16706.301,E2 -16706.301} C_VEL
LIN {X 0,Y 291.38,Z 309.187,A -85,B 0,C 180,E1 -16710.261,E2 -16710.261} C_VEL
LIN {X 0,Y 291.411,Z 309.184,A -85,B 0,C 180,E1 -16714.272,E2 -16714.272} C_VEL
LIN {X 0,Y 291.385,Z 309.187,A -85,B 0,C 180,E1 -16717.3,E2 -16717.3} C_VEL
LIN {X 0,Y 291.454,Z 309.171,A -85,B 0,C 180,E1 -16720.27,E2 -16720.27} C_VEL
LIN {X 0,Y 291.551,Z 309.163,A -85,B 0,C 180,E1 -16724.624,E2 -16724.624} C_VEL
LIN {X 0,Y 291.533,Z 309.167,A -85,B 0,C 180,E1 -16728.881,E2 -16728.881} C_VEL
LIN {X 0,Y 291.705,Z 309.14,A -85,B 0,C 180,E1 -16731.689,E2 -16731.689} C_VEL
LIN {X 0,Y 291.628,Z 309.159,A -85,B 0,C 180,E1 -16734.469,E2 -16734.469} C_VEL
LIN {X 0,Y 291.887,Z 309.126,A -85,B 0,C 180,E1 -16738.621,E2 -16738.621} C_VEL
LIN {X 0,Y 291.887,Z 309.121,A -85,B 0,C 180,E1 -16741.38,E2 -16741.38} C_VEL
LIN {X 0,Y 291.743,Z 309.144,A -85,B 0,C 180,E1 -16746.918,E2 -16746.918} C_VEL
LIN {X 0,Y 291.626,Z 309.152,A -85,B 0,C 180,E1 -16749.712,E2 -16749.712} C_VEL
LIN {X 0,Y 291.519,Z 309.166,A -85,B 0,C 180,E1 -16753.951,E2 -16753.951} C_VEL
LIN {X 0,Y 291.484,Z 309.172,A -85,B 0,C 180,E1 -16756.819,E2 -16756.819} C_VEL
LIN {X 0,Y 291.448,Z 309.179,A -85,B 0,C 180,E1 -16759.876,E2 -16759.876} C_VEL
LIN {X 0,Y 291.398,Z 309.185,A -85,B 0,C 180,E1 -16764.206,E2 -16764.206} C_VEL
LIN {X 0,Y 291.418,Z 309.186,A -85,B 0,C 180,E1 -16767.273,E2 -16767.273} C_VEL
LIN {X 0,Y 291.332,Z 309.194,A -85,B 0,C 180,E1 -16770.438,E2 -16770.438} C_VEL
LIN {X 0,Y 291.343,Z 309.193,A -85,B 0,C 180,E1 -16773.699,E2 -16773.699} C_VEL
LIN {X 0,Y 291.368,Z 309.189,A -85,B 0,C 180,E1 -16777.253,E2 -16777.253} C_VEL
LIN {X 0,Y 291.329,Z 309.192,A -85,B 0,C 180,E1 -16780.644,E2 -16780.644} C_VEL
LIN {X 0,Y 291.289,Z 309.201,A -85,B 0,C 180,E1 -16784.403,E2 -16784.403} C_VEL
LIN {X 0,Y 291.294,Z 309.201,A -85,B 0,C 180,E1 -16788.412,E2 -16788.412} C_VEL
LIN {X 0,Y 291.308,Z 309.308,A -85,B 0,C 180,E1 -16790.167,E2 -16790.167} C_VEL
LIN {X 0,Y 291.651,Z 310.648,A -85,B 0,C 180,E1 -16790.655,E2 -16790.655} C_VEL
LIN {X 0,Y 300.51,Z 327.304,A -85,B 0,C 180,E1 -16792.264,E2 -16792.264} C_VEL
LIN {X 0,Y 307.448,Z 342.352,A -85,B 0,C 180,E1 -16793.493,E2 -16793.493} C_VEL
LIN {X 0,Y 309.515,Z 347.181,A -85,B 0,C 180,E1 -16793.854,E2 -16793.854} C_VEL
LIN {X 0,Y 307.262,Z 417.17,A -85,B 0,C 180,E1 -16795.495,E2 -16795.495} C_VEL
LIN {X 0,Y 306.522,Z 430.337,A -85,B 0,C 180,E1 -16796.065,E2 -16796.065} C_VEL
LIN {X 0,Y 305.256,Z 442.887,A -85,B 0,C 180,E1 -16796.853,E2 -16796.853} C_VEL
LIN {X 0,Y 303.717,Z 454.508,A -85,B 0,C 180,E1 -16797.845,E2 -16797.845} C_VEL
LIN {X 0,Y 302.097,Z 465.059,A -85,B 0,C 180,E1 -16799.022,E2 -16799.022} C_VEL
LIN {X 0,Y 300.209,Z 475.899,A -85,B 0,C 180,E1 -16800.554,E2 -16800.554} C_VEL
LIN {X 0,Y 298.239,Z 485.605,A -85,B 0,C 180,E1 -16802.264,E2 -16802.264} C_VEL
LIN {X 0,Y 296.472,Z 493.444,A -85,B 0,C 180,E1 -16803.977,E2 -16803.977} C_VEL
LIN {X 0,Y 294.618,Z 501.14,A -85,B 0,C 180,E1 -16806.077,E2 -16806.077} C_VEL
LIN {X 0,Y 293.093,Z 507.249,A -85,B 0,C 180,E1 -16808.182,E2 -16808.182} C_VEL
LIN {X 0,Y 291.886,Z 512.048,A -85,B 0,C 180,E1 -16810.301,E2 -16810.301} C_VEL
LIN {X 0,Y 290.981,Z 515.692,A -85,B 0,C 180,E1 -16812.429,E2 -16812.429} C_VEL
LIN {X 0,Y 290.342,Z 518.286,A -85,B 0,C 180,E1 -16814.559,E2 -16814.559} C_VEL
LIN {X 0,Y 290.037,Z 519.493,A -85,B 0,C 180,E1 -16815.978,E2 -16815.978} C_VEL
LIN {X 0,Y 289.753,Z 520.261,A -85,B 0,C 180,E1 -16817.392,E2 -16817.392} C_VEL
LIN {X 0,Y 289.464,Z 520.583,A -85,B 0,C 180,E1 -16820.216,E2 -16820.216} C_VEL
LIN {X 0,Y 289.503,Z 520.162,A -85,B 0,C 180,E1 -16821.626,E2 -16821.626} C_VEL
LIN {X 0,Y 289.677,Z 518.381,A -85,B 0,C 180,E1 -16824.118,E2 -16824.118} C_VEL
LIN {X 0,Y 289.848,Z 515.41,A -85,B 0,C 180,E1 -16826.526,E2 -16826.526} C_VEL
LIN {X 0,Y 290.3,Z 511.754,A -85,B 0,C 180,E1 -16828.614,E2 -16828.614} C_VEL
LIN {X 0,Y 290.783,Z 507.007,A -85,B 0,C 180,E1 -16830.693,E2 -16830.693} C_VEL
LIN {X 0,Y 291.783,Z 499.892,A -85,B 0,C 180,E1 -16833.107,E2 -16833.107} C_VEL
LIN {X 0,Y 292.881,Z 492.128,A -85,B 0,C 180,E1 -16835.164,E2 -16835.164} C_VEL
LIN {X 0,Y 294.211,Z 482.444,A -85,B 0,C 180,E1 -16837.205,E2 -16837.205} C_VEL
LIN {X 0,Y 295.584,Z 472.393,A -85,B 0,C 180,E1 -16838.891,E2 -16838.891} C_VEL
LIN {X 0,Y 296.964,Z 461.013,A -85,B 0,C 180,E1 -16840.397,E2 -16840.397} C_VEL
LIN {X 0,Y 298.085,Z 449.861,A -85,B 0,C 180,E1 -16841.562,E2 -16841.562} C_VEL
LIN {X 0,Y 299.033,Z 437.334,A -85,B 0,C 180,E1 -16842.557,E2 -16842.557} C_VEL
LIN {X 0,Y 299.852,Z 423.888,A -85,B 0,C 180,E1 -16843.297,E2 -16843.297} C_VEL
LIN {X 0,Y 300.249,Z 411.4,A -85,B 0,C 180,E1 -16843.73,E2 -16843.73} C_VEL
LIN {X 0,Y 301.969,Z 338.21,A -85,B 0,C 180,E1 -16845.442,E2 -16845.442} C_VEL
LIN {X 0,Y 295.854,Z 320.471,A -85,B 0,C 180,E1 -16846.362,E2 -16846.362} C_VEL
LIN {X 0,Y 291.54,Z 309.57,A -85,B 0,C 180,E1 -16847.018,E2 -16847.018} C_VEL
LIN {X 0,Y 291.46,Z 309.181,A -85,B 0,C 180,E1 -16847.244,E2 -16847.244} C_VEL
LIN {X 0,Y 291.429,Z 309.182,A -85,B 0,C 180,E1 -16849.861,E2 -16849.861} C_VEL
LIN {X 0,Y 291.364,Z 309.186,A -85,B 0,C 180,E1 -16854.209,E2 -16854.209} C_VEL
LIN {X 0,Y 291.357,Z 309.19,A -85,B 0,C 180,E1 -16857.279,E2 -16857.279} C_VEL
LIN {X 0,Y 291.323,Z 309.194,A -85,B 0,C 180,E1 -16860.439,E2 -16860.439} C_VEL
LIN {X 0,Y 291.349,Z 309.191,A -85,B 0,C 180,E1 -16863.699,E2 -16863.699} C_VEL
LIN {X 0,Y 291.364,Z 309.193,A -85,B 0,C 180,E1 -16867.25,E2 -16867.25} C_VEL
LIN {X 0,Y 291.305,Z 309.195,A -85,B 0,C 180,E1 -16870.648,E2 -16870.648} C_VEL
LIN {X 0,Y 291.286,Z 309.198,A -85,B 0,C 180,E1 -16874.404,E2 -16874.404} C_VEL
LIN {X 0,Y 291.299,Z 309.192,A -85,B 0,C 180,E1 -16878.412,E2 -16878.412} C_VEL
LIN {X 0,Y 291.402,Z 309.184,A -85,B 0,C 180,E1 -16882.918,E2 -16882.918} C_VEL
LIN {X 0,Y 291.348,Z 309.186,A -85,B 0,C 180,E1 -16886.301,E2 -16886.301} C_VEL
LIN {X 0,Y 291.368,Z 309.189,A -85,B 0,C 180,E1 -16890.245,E2 -16890.245} C_VEL
LIN {X 0,Y 290.775,Z 309.265,A -85,B 0,C 180,E1 -16891.398,E2 -16891.398} C_VEL
LIN {X 0,Y 287.917,Z 309.621,A -85,B 0,C 180,E1 -16893.274,E2 -16893.274} C_VEL
LIN {X 0,Y 285.449,Z 309.927,A -85,B 0,C 180,E1 -16894.798,E2 -16894.798} C_VEL
LIN {X 0,Y 284.396,Z 310.056,A -85,B 0,C 180,E1 -16895.98,E2 -16895.98} C_VEL
LIN {X 0,Y 284.317,Z 310.064,A -85,B 0,C 180,E1 -16896.38,E2 -16896.38} C_VEL
LIN {X 0,Y 284.381,Z 310.063,A -85,B 0,C 180,E1 -16899.904,E2 -16899.904} C_VEL
LIN {X 0,Y 284.453,Z 310.04,A -85,B 0,C 180,E1 -16904.492,E2 -16904.492} C_VEL
LIN {X 0,Y 284.486,Z 310.046,A -85,B 0,C 180,E1 -16908.601,E2 -16908.601} C_VEL
LIN {X 0,Y 284.613,Z 310.029,A -85,B 0,C 180,E1 -16911.479,E2 -16911.479} C_VEL
LIN {X 0,Y 284.572,Z 310.027,A -85,B 0,C 180,E1 -16914.33,E2 -16914.33} C_VEL
LIN {X 0,Y 284.842,Z 310.002,A -85,B 0,C 180,E1 -16918.586,E2 -16918.586} C_VEL
LIN {X 0,Y 284.847,Z 310,A -85,B 0,C 180,E1 -16921.413,E2 -16921.413} C_VEL
LIN {X 0,Y 284.645,Z 310.019,A -85,B 0,C 180,E1 -16927.091,E2 -16927.091} C_VEL
LIN {X 0,Y 284.518,Z 310.041,A -85,B 0,C 180,E1 -16929.957,E2 -16929.957} C_VEL
LIN {X 0,Y 284.467,Z 310.049,A -85,B 0,C 180,E1 -16934.303,E2 -16934.303} C_VEL
LIN {X 0,Y 284.337,Z 310.067,A -85,B 0,C 180,E1 -16938.743,E2 -16938.743} C_VEL
LIN {X 0,Y 284.331,Z 310.066,A -85,B 0,C 180,E1 -16943.296,E2 -16943.296} C_VEL
LIN {X 0,Y 284.331,Z 310.068,A -85,B 0,C 180,E1 -16947.145,E2 -16947.145} C_VEL
LIN {X 0,Y 284.282,Z 310.074,A -85,B 0,C 180,E1 -16951.276,E2 -16951.276} C_VEL
LIN {X 0,Y 284.339,Z 310.068,A -85,B 0,C 180,E1 -16955.346,E2 -16955.346} C_VEL
LIN {X 0,Y 284.3,Z 310.07,A -85,B 0,C 180,E1 -16958.171,E2 -16958.171} C_VEL
LIN {X 0,Y 284.24,Z 310.077,A -85,B 0,C 180,E1 -16962.116,E2 -16962.116} C_VEL
LIN {X 0,Y 284.24,Z 310.076,A -85,B 0,C 180,E1 -16966.185,E2 -16966.185} C_VEL
LIN {X 0,Y 284.285,Z 310.072,A -85,B 0,C 180,E1 -16970.029,E2 -16970.029} C_VEL
LIN {X 0,Y 284.33,Z 310.071,A -85,B 0,C 180,E1 -16973.613,E2 -16973.613} C_VEL
LIN {X 0,Y 284.346,Z 310.223,A -85,B 0,C 180,E1 -16976.531,E2 -16976.531} C_VEL
LIN {X 0,Y 286.624,Z 320.737,A -85,B 0,C 180,E1 -16979.844,E2 -16979.844} C_VEL
LIN {X 0,Y 288.471,Z 330.639,A -85,B 0,C 180,E1 -16982.818,E2 -16982.818} C_VEL
LIN {X 0,Y 288.438,Z 333.938,A -85,B 0,C 180,E1 -16983.743,E2 -16983.743} C_VEL
LIN {X 0,Y 292.326,Z 362.357,A -85,B 0,C 180,E1 -16984.814,E2 -16984.814} C_VEL
LIN {X 0,Y 294.547,Z 382.324,A -85,B 0,C 180,E1 -16985.497,E2 -16985.497} C_VEL
LIN {X 0,Y 293.172,Z 442.822,A -85,B 0,C 180,E1 -16986.979,E2 -16986.979} C_VEL
LIN {X 0,Y 292.278,Z 456.137,A -85,B 0,C 180,E1 -16987.559,E2 -16987.559} C_VEL
LIN {X 0,Y 291.173,Z 468.933,A -85,B 0,C 180,E1 -16988.401,E2 -16988.401} C_VEL
LIN {X 0,Y 289.873,Z 480.273,A -85,B 0,C 180,E1 -16989.417,E2 -16989.417} C_VEL
LIN {X 0,Y 288.375,Z 491.999,A -85,B 0,C 180,E1 -16990.79,E2 -16990.79} C_VEL
LIN {X 0,Y 287,Z 502.556,A -85,B 0,C 180,E1 -16992.359,E2 -16992.359} C_VEL
LIN {X 0,Y 285.848,Z 511.752,A -85,B 0,C 180,E1 -16994.059,E2 -16994.059} C_VEL
LIN {X 0,Y 284.597,Z 520.51,A -85,B 0,C 180,E1 -16996.067,E2 -16996.067} C_VEL
LIN {X 0,Y 283.53,Z 527.986,A -85,B 0,C 180,E1 -16998.199,E2 -16998.199} C_VEL
LIN {X 0,Y 282.862,Z 534.868,A -85,B 0,C 180,E1 -17000.705,E2 -17000.705} C_VEL
LIN {X 0,Y 282.568,Z 539.396,A -85,B 0,C 180,E1 -17002.855,E2 -17002.855} C_VEL
LIN {X 0,Y 282.463,Z 541.962,A -85,B 0,C 180,E1 -17004.409,E2 -17004.409} C_VEL
LIN {X 0,Y 282.458,Z 545.234,A -85,B 0,C 180,E1 -17007.147,E2 -17007.147} C_VEL
LIN {X 0,Y 282.454,Z 546.285,A -85,B 0,C 180,E1 -17008.573,E2 -17008.573} C_VEL
LIN {X 0,Y 282.495,Z 546.94,A -85,B 0,C 180,E1 -17009.999,E2 -17009.999} C_VEL
LIN {X 0,Y 282.43,Z 547.198,A -85,B 0,C 180,E1 -17011.425,E2 -17011.425} C_VEL
LIN {X 0,Y 282.429,Z 547.063,A -85,B 0,C 180,E1 -17012.852,E2 -17012.852} C_VEL
LIN {X 0,Y 282.408,Z 545.723,A -85,B 0,C 180,E1 -17015.474,E2 -17015.474} C_VEL
LIN {X 0,Y 282.505,Z 544.176,A -85,B 0,C 180,E1 -17017.144,E2 -17017.144} C_VEL
LIN {X 0,Y 282.952,Z 541.342,A -85,B 0,C 180,E1 -17019.29,E2 -17019.29} C_VEL
LIN {X 0,Y 283.65,Z 537.498,A -85,B 0,C 180,E1 -17021.432,E2 -17021.432} C_VEL
LIN {X 0,Y 284.713,Z 532.552,A -85,B 0,C 180,E1 -17023.561,E2 -17023.561} C_VEL
LIN {X 0,Y 286.252,Z 526.357,A -85,B 0,C 180,E1 -17025.667,E2 -17025.667} C_VEL
LIN {X 0,Y 287.916,Z 519.15,A -85,B 0,C 180,E1 -17027.641,E2 -17027.641} C_VEL
LIN {X 0,Y 289.735,Z 510.839,A -85,B 0,C 180,E1 -17029.482,E2 -17029.482} C_VEL
LIN {X 0,Y 292.129,Z 500.231,A -85,B 0,C 180,E1 -17031.337,E2 -17031.337} C_VEL
LIN {X 0,Y 294.299,Z 489.452,A -85,B 0,C 180,E1 -17032.833,E2 -17032.833} C_VEL
LIN {X 0,Y 296.247,Z 478.956,A -85,B 0,C 180,E1 -17033.969,E2 -17033.969} C_VEL
LIN {X 0,Y 297.988,Z 467.474,A -85,B 0,C 180,E1 -17034.933,E2 -17034.933} C_VEL
LIN {X 0,Y 299.508,Z 454.545,A -85,B 0,C 180,E1 -17035.727,E2 -17035.727} C_VEL
LIN {X 0,Y 300.527,Z 442.005,A -85,B 0,C 180,E1 -17036.239,E2 -17036.239} C_VEL
LIN {X 0,Y 302.373,Z 383.406,A -85,B 0,C 180,E1 -17037.655,E2 -17037.655} C_VEL
LIN {X 0,Y 298.661,Z 360.312,A -85,B 0,C 180,E1 -17038.723,E2 -17038.723} C_VEL
LIN {X 0,Y 295.527,Z 345.542,A -85,B 0,C 180,E1 -17039.521,E2 -17039.521} C_VEL
LIN {X 0,Y 290.736,Z 335.022,A -85,B 0,C 180,E1 -17040.436,E2 -17040.436} C_VEL
LIN {X 0,Y 289.929,Z 332.84,A -85,B 0,C 180,E1 -17040.646,E2 -17040.646} C_VEL
LIN {X 0,Y 287.279,Z 321.088,A -85,B 0,C 180,E1 -17044.664,E2 -17044.664} C_VEL
LIN {X 0,Y 284.784,Z 311.84,A -85,B 0,C 180,E1 -17048.093,E2 -17048.093} C_VEL
LIN {X 0,Y 284.306,Z 310.07,A -85,B 0,C 180,E1 -17048.848,E2 -17048.848} C_VEL
LIN {X 0,Y 284.266,Z 310.074,A -85,B 0,C 180,E1 -17052.124,E2 -17052.124} C_VEL
LIN {X 0,Y 284.251,Z 310.074,A -85,B 0,C 180,E1 -17056.189,E2 -17056.189} C_VEL
LIN {X 0,Y 284.303,Z 310.068,A -85,B 0,C 180,E1 -17060.023,E2 -17060.023} C_VEL
LIN {X 0,Y 284.329,Z 310.066,A -85,B 0,C 180,E1 -17063.614,E2 -17063.614} C_VEL
LIN {X 0,Y 284.303,Z 310.067,A -85,B 0,C 180,E1 -17067.189,E2 -17067.189} C_VEL
LIN {X 0,Y 284.351,Z 310.063,A -85,B 0,C 180,E1 -17070.375,E2 -17070.375} C_VEL
LIN {X 0,Y 284.372,Z 310.059,A -85,B 0,C 180,E1 -17073.586,E2 -17073.586} C_VEL
LIN {X 0,Y 284.365,Z 310.057,A -85,B 0,C 180,E1 -17076.707,E2 -17076.707} C_VEL
LIN {X 0,Y 284.4,Z 310.059,A -85,B 0,C 180,E1 -17081.262,E2 -17081.262} C_VEL
LIN {X 0,Y 284.488,Z 310.041,A -85,B 0,C 180,E1 -17084.459,E2 -17084.459} C_VEL
LIN {X 0,Y 284.485,Z 310.042,A -85,B 0,C 180,E1 -17088.602,E2 -17088.602} C_VEL
LIN {X 0,Y 284.655,Z 310.019,A -85,B 0,C 180,E1 -17091.481,E2 -17091.481} C_VEL
LIN {X 0,Y 284.598,Z 310.034,A -85,B 0,C 180,E1 -17094.332,E2 -17094.332} C_VEL
LIN {X 0,Y 284.853,Z 310.002,A -85,B 0,C 180,E1 -17098.587,E2 -17098.587} C_VEL
LIN {X 0,Y 284.853,Z 309.997,A -85,B 0,C 180,E1 -17101.414,E2 -17101.414} C_VEL
LIN {X 0,Y 284.695,Z 310.023,A -85,B 0,C 180,E1 -17107.091,E2 -17107.091} C_VEL
LIN {X 0,Y 284.563,Z 310.033,A -85,B 0,C 180,E1 -17109.956,E2 -17109.956} C_VEL
LIN {X 0,Y 284.479,Z 310.043,A -85,B 0,C 180,E1 -17114.303,E2 -17114.303} C_VEL
LIN {X 0,Y 284.422,Z 310.049,A -85,B 0,C 180,E1 -17117.249,E2 -17117.249} C_VEL
LIN {X 0,Y 284.376,Z 310.06,A -85,B 0,C 180,E1 -17120.243,E2 -17120.243} C_VEL
LIN {X 0,Y 284.367,Z 310.061,A -85,B 0,C 180,E1 -17123.876,E2 -17123.876} C_VEL
LIN {X 0,Y 284.393,Z 310.062,A -85,B 0,C 180,E1 -17127.174,E2 -17127.174} C_VEL
LIN {X 0,Y 284.292,Z 310.069,A -85,B 0,C 180,E1 -17131.275,E2 -17131.275} C_VEL
LIN {X 0,Y 284.339,Z 310.06,A -85,B 0,C 180,E1 -17135.349,E2 -17135.349} C_VEL
LIN {X 0,Y 284.304,Z 310.063,A -85,B 0,C 180,E1 -17138.171,E2 -17138.171} C_VEL
LIN {X 0,Y 284.267,Z 310.075,A -85,B 0,C 180,E1 -17142.125,E2 -17142.125} C_VEL
LIN {X 0,Y 284.237,Z 310.078,A -85,B 0,C 180,E1 -17146.187,E2 -17146.187} C_VEL
LIN {X 0,Y 284.253,Z 310.113,A -85,B 0,C 180,E1 -17149.332,E2 -17149.332} C_VEL
LIN {X 0,Y 284.511,Z 311.244,A -85,B 0,C 180,E1 -17149.686,E2 -17149.686} C_VEL
LIN {X 0,Y 286.442,Z 314.675,A -85,B 0,C 180,E1 -17150.062,E2 -17150.062} C_VEL
LIN {X 0,Y 294.893,Z 330.409,A -85,B 0,C 180,E1 -17151.651,E2 -17151.651} C_VEL
LIN {X 0,Y 301.817,Z 345.461,A -85,B 0,C 180,E1 -17152.924,E2 -17152.924} C_VEL
LIN {X 0,Y 303.435,Z 349.255,A -85,B 0,C 180,E1 -17153.218,E2 -17153.218} C_VEL
LIN {X 0,Y 301.099,Z 417.16,A -85,B 0,C 180,E1 -17154.83,E2 -17154.83} C_VEL
LIN {X 0,Y 300.35,Z 429.955,A -85,B 0,C 180,E1 -17155.381,E2 -17155.381} C_VEL
LIN {X 0,Y 299.098,Z 442.588,A -85,B 0,C 180,E1 -17156.181,E2 -17156.181} C_VEL
LIN {X 0,Y 297.606,Z 453.468,A -85,B 0,C 180,E1 -17157.103,E2 -17157.103} C_VEL
LIN {X 0,Y 295.879,Z 464.349,A -85,B 0,C 180,E1 -17158.297,E2 -17158.297} C_VEL
LIN {X 0,Y 293.929,Z 475.384,A -85,B 0,C 180,E1 -17159.861,E2 -17159.861} C_VEL
LIN {X 0,Y 291.794,Z 485.231,A -85,B 0,C 180,E1 -17161.597,E2 -17161.597} C_VEL
LIN {X 0,Y 289.863,Z 493.551,A -85,B 0,C 180,E1 -17163.428,E2 -17163.428} C_VEL
LIN {X 0,Y 287.998,Z 501.032,A -85,B 0,C 180,E1 -17165.491,E2 -17165.491} C_VEL
LIN {X 0,Y 286.345,Z 507.225,A -85,B 0,C 180,E1 -17167.641,E2 -17167.641} C_VEL
LIN {X 0,Y 285.069,Z 512.101,A -85,B 0,C 180,E1 -17169.81,E2 -17169.81} C_VEL
LIN {X 0,Y 284.056,Z 515.817,A -85,B 0,C 180,E1 -17171.986,E2 -17171.986} C_VEL
LIN {X 0,Y 283.358,Z 518.478,A -85,B 0,C 180,E1 -17174.168,E2 -17174.168} C_VEL
LIN {X 0,Y 283.028,Z 519.717,A -85,B 0,C 180,E1 -17175.623,E2 -17175.623} C_VEL
LIN {X 0,Y 282.712,Z 520.546,A -85,B 0,C 180,E1 -17177.073,E2 -17177.073} C_VEL
LIN {X 0,Y 282.382,Z 520.932,A -85,B 0,C 180,E1 -17179.968,E2 -17179.968} C_VEL
LIN {X 0,Y 282.393,Z 520.543,A -85,B 0,C 180,E1 -17181.413,E2 -17181.413} C_VEL
LIN {X 0,Y 282.605,Z 518.689,A -85,B 0,C 180,E1 -17184.131,E2 -17184.131} C_VEL
LIN {X 0,Y 282.763,Z 515.946,A -85,B 0,C 180,E1 -17186.438,E2 -17186.438} C_VEL
LIN {X 0,Y 283.22,Z 512.359,A -85,B 0,C 180,E1 -17188.579,E2 -17188.579} C_VEL
LIN {X 0,Y 283.709,Z 507.686,A -85,B 0,C 180,E1 -17190.711,E2 -17190.711} C_VEL
LIN {X 0,Y 284.719,Z 500.653,A -85,B 0,C 180,E1 -17193.185,E2 -17193.185} C_VEL
LIN {X 0,Y 285.843,Z 493.03,A -85,B 0,C 180,E1 -17195.291,E2 -17195.291} C_VEL
LIN {X 0,Y 287.216,Z 483.46,A -85,B 0,C 180,E1 -17197.382,E2 -17197.382} C_VEL
LIN {X 0,Y 288.607,Z 473.587,A -85,B 0,C 180,E1 -17199.108,E2 -17199.108} C_VEL
LIN {X 0,Y 290.011,Z 462.448,A -85,B 0,C 180,E1 -17200.649,E2 -17200.649} C_VEL
LIN {X 0,Y 291.214,Z 451.546,A -85,B 0,C 180,E1 -17201.838,E2 -17201.838} C_VEL
LIN {X 0,Y 292.155,Z 439.538,A -85,B 0,C 180,E1 -17202.858,E2 -17202.858} C_VEL
LIN {X 0,Y 293.028,Z 427.035,A -85,B 0,C 180,E1 -17203.613,E2 -17203.613} C_VEL
LIN {X 0,Y 293.513,Z 413.267,A -85,B 0,C 180,E1 -17204.143,E2 -17204.143} C_VEL
LIN {X 0,Y 295.344,Z 339.507,A -85,B 0,C 180,E1 -17205.911,E2 -17205.911} C_VEL
LIN {X 0,Y 289.014,Z 321.544,A -85,B 0,C 180,E1 -17206.888,E2 -17206.888} C_VEL
LIN {X 0,Y 284.576,Z 310.809,A -85,B 0,C 180,E1 -17207.552,E2 -17207.552} C_VEL
LIN {X 0,Y 284.429,Z 310.056,A -85,B 0,C 180,E1 -17207.62,E2 -17207.62} C_VEL
LIN {X 0,Y 284.372,Z 310.062,A -85,B 0,C 180,E1 -17210.244,E2 -17210.244} C_VEL
LIN {X 0,Y 284.326,Z 310.062,A -85,B 0,C 180,E1 -17213.854,E2 -17213.854} C_VEL
LIN {X 0,Y 284.288,Z 310.068,A -85,B 0,C 180,E1 -17218.016,E2 -17218.016} C_VEL
LIN {X 0,Y 284.29,Z 310.073,A -85,B 0,C 180,E1 -17221.276,E2 -17221.276} C_VEL
LIN {X 0,Y 284.342,Z 310.067,A -85,B 0,C 180,E1 -17225.347,E2 -17225.347} C_VEL
LIN {X 0,Y 284.303,Z 310.068,A -85,B 0,C 180,E1 -17228.172,E2 -17228.172} C_VEL
LIN {X 0,Y 284.242,Z 310.073,A -85,B 0,C 180,E1 -17232.117,E2 -17232.117} C_VEL
LIN {X 0,Y 284.242,Z 310.072,A -85,B 0,C 180,E1 -17236.186,E2 -17236.186} C_VEL
LIN {X 0,Y 284.26,Z 310.073,A -85,B 0,C 180,E1 -17240.036,E2 -17240.036} C_VEL
LIN {X 0,Y 284.33,Z 310.063,A -85,B 0,C 180,E1 -17243.613,E2 -17243.613} C_VEL
LIN {X 0,Y 284.311,Z 310.064,A -85,B 0,C 180,E1 -17247.19,E2 -17247.19} C_VEL
LIN {X 0,Y 284.342,Z 310.064,A -85,B 0,C 180,E1 -17250.374,E2 -17250.374} C_VEL
LIN {X 0,Y 284.304,Z 310.065,A -85,B 0,C 180,E1 -17253.579,E2 -17253.579} C_VEL
LIN {X 0,Y 284.317,Z 310.064,A -85,B 0,C 180,E1 -17256.38,E2 -17256.38} C_VEL
LIN {X 0,Y 283.672,Z 310.149,A -85,B 0,C 180,E1 -17257.563,E2 -17257.563} C_VEL
LIN {X 0,Y 280.85,Z 310.5,A -85,B 0,C 180,E1 -17259.491,E2 -17259.491} C_VEL
LIN {X 0,Y 278.444,Z 310.799,A -85,B 0,C 180,E1 -17261.056,E2 -17261.056} C_VEL
LIN {X 0,Y 277.41,Z 310.924,A -85,B 0,C 180,E1 -17262.269,E2 -17262.269} C_VEL
LIN {X 0,Y 277.325,Z 310.931,A -85,B 0,C 180,E1 -17262.679,E2 -17262.679} C_VEL
LIN {X 0,Y 277.415,Z 310.915,A -85,B 0,C 180,E1 -17265.324,E2 -17265.324} C_VEL
LIN {X 0,Y 277.462,Z 310.922,A -85,B 0,C 180,E1 -17269.787,E2 -17269.787} C_VEL
LIN {X 0,Y 277.605,Z 310.899,A -85,B 0,C 180,E1 -17272.727,E2 -17272.727} C_VEL
LIN {X 0,Y 277.809,Z 310.879,A -85,B 0,C 180,E1 -17278.55,E2 -17278.55} C_VEL
LIN {X 0,Y 277.813,Z 310.876,A -85,B 0,C 180,E1 -17281.449,E2 -17281.449} C_VEL
LIN {X 0,Y 277.604,Z 310.895,A -85,B 0,C 180,E1 -17287.272,E2 -17287.272} C_VEL
LIN {X 0,Y 277.459,Z 310.922,A -85,B 0,C 180,E1 -17290.213,E2 -17290.213} C_VEL
LIN {X 0,Y 277.413,Z 310.93,A -85,B 0,C 180,E1 -17294.675,E2 -17294.675} C_VEL
LIN {X 0,Y 277.289,Z 310.943,A -85,B 0,C 180,E1 -17299.238,E2 -17299.238} C_VEL
LIN {X 0,Y 277.285,Z 310.943,A -85,B 0,C 180,E1 -17303.924,E2 -17303.924} C_VEL
LIN {X 0,Y 277.269,Z 310.946,A -85,B 0,C 180,E1 -17307.481,E2 -17307.481} C_VEL
LIN {X 0,Y 277.241,Z 310.949,A -85,B 0,C 180,E1 -17312.164,E2 -17312.164} C_VEL
LIN {X 0,Y 277.276,Z 310.945,A -85,B 0,C 180,E1 -17315.796,E2 -17315.796} C_VEL
LIN {X 0,Y 277.219,Z 310.955,A -85,B 0,C 180,E1 -17319.33,E2 -17319.33} C_VEL
LIN {X 0,Y 277.193,Z 310.959,A -85,B 0,C 180,E1 -17323.201,E2 -17323.201} C_VEL
LIN {X 0,Y 277.194,Z 310.958,A -85,B 0,C 180,E1 -17327.33,E2 -17327.33} C_VEL
LIN {X 0,Y 277.258,Z 310.95,A -85,B 0,C 180,E1 -17331.794,E2 -17331.794} C_VEL
LIN {X 0,Y 277.29,Z 310.947,A -85,B 0,C 180,E1 -17336.027,E2 -17336.027} C_VEL
LIN {X 0,Y 279.814,Z 322.755,A -85,B 0,C 180,E1 -17339.844,E2 -17339.844} C_VEL
LIN {X 0,Y 281.612,Z 332.713,A -85,B 0,C 180,E1 -17342.905,E2 -17342.905} C_VEL
LIN {X 0,Y 281.662,Z 334.01,A -85,B 0,C 180,E1 -17343.193,E2 -17343.193} C_VEL
LIN {X 0,Y 285.674,Z 362.415,A -85,B 0,C 180,E1 -17344.292,E2 -17344.292} C_VEL
LIN {X 0,Y 287.916,Z 382.264,A -85,B 0,C 180,E1 -17344.995,E2 -17344.995} C_VEL
LIN {X 0,Y 286.462,Z 443.012,A -85,B 0,C 180,E1 -17346.522,E2 -17346.522} C_VEL
LIN {X 0,Y 285.531,Z 456.629,A -85,B 0,C 180,E1 -17347.142,E2 -17347.142} C_VEL
LIN {X 0,Y 284.447,Z 468.643,A -85,B 0,C 180,E1 -17347.959,E2 -17347.959} C_VEL
LIN {X 0,Y 282.99,Z 480.767,A -85,B 0,C 180,E1 -17349.083,E2 -17349.083} C_VEL
LIN {X 0,Y 281.453,Z 492.343,A -85,B 0,C 180,E1 -17350.489,E2 -17350.489} C_VEL
LIN {X 0,Y 280.039,Z 502.783,A -85,B 0,C 180,E1 -17352.095,E2 -17352.095} C_VEL
LIN {X 0,Y 278.952,Z 510.75,A -85,B 0,C 180,E1 -17353.603,E2 -17353.603} C_VEL
LIN {X 0,Y 277.649,Z 519.847,A -85,B 0,C 180,E1 -17355.711,E2 -17355.711} C_VEL
LIN {X 0,Y 276.552,Z 527.383,A -85,B 0,C 180,E1 -17357.897,E2 -17357.897} C_VEL
LIN {X 0,Y 275.819,Z 534.339,A -85,B 0,C 180,E1 -17360.466,E2 -17360.466} C_VEL
LIN {X 0,Y 275.499,Z 538.914,A -85,B 0,C 180,E1 -17362.671,E2 -17362.671} C_VEL
LIN {X 0,Y 275.373,Z 541.803,A -85,B 0,C 180,E1 -17364.47,E2 -17364.47} C_VEL
LIN {X 0,Y 275.384,Z 544.827,A -85,B 0,C 180,E1 -17367.073,E2 -17367.073} C_VEL
LIN {X 0,Y 275.373,Z 545.907,A -85,B 0,C 180,E1 -17368.537,E2 -17368.537} C_VEL
LIN {X 0,Y 275.411,Z 546.58,A -85,B 0,C 180,E1 -17369.999,E2 -17369.999} C_VEL
LIN {X 0,Y 275.35,Z 546.858,A -85,B 0,C 180,E1 -17371.462,E2 -17371.462} C_VEL
LIN {X 0,Y 275.354,Z 546.749,A -85,B 0,C 180,E1 -17372.925,E2 -17372.925} C_VEL
LIN {X 0,Y 275.331,Z 545.597,A -85,B 0,C 180,E1 -17375.437,E2 -17375.437} C_VEL
LIN {X 0,Y 275.455,Z 543.931,A -85,B 0,C 180,E1 -17377.328,E2 -17377.328} C_VEL
LIN {X 0,Y 275.921,Z 541.137,A -85,B 0,C 180,E1 -17379.529,E2 -17379.529} C_VEL
LIN {X 0,Y 276.64,Z 537.337,A -85,B 0,C 180,E1 -17381.725,E2 -17381.725} C_VEL
LIN {X 0,Y 277.804,Z 532.438,A -85,B 0,C 180,E1 -17383.905,E2 -17383.905} C_VEL
LIN {X 0,Y 279.384,Z 526.293,A -85,B 0,C 180,E1 -17386.063,E2 -17386.063} C_VEL
LIN {X 0,Y 281.304,Z 518.26,A -85,B 0,C 180,E1 -17388.309,E2 -17388.309} C_VEL
LIN {X 0,Y 283.467,Z 509.158,A -85,B 0,C 180,E1 -17390.309,E2 -17390.309} C_VEL
LIN {X 0,Y 285.752,Z 499.353,A -85,B 0,C 180,E1 -17392.028,E2 -17392.028} C_VEL
LIN {X 0,Y 288.089,Z 488.423,A -85,B 0,C 180,E1 -17393.544,E2 -17393.544} C_VEL
LIN {X 0,Y 290.065,Z 477.736,A -85,B 0,C 180,E1 -17394.704,E2 -17394.704} C_VEL
LIN {X 0,Y 292.021,Z 464.889,A -85,B 0,C 180,E1 -17395.766,E2 -17395.766} C_VEL
LIN {X 0,Y 293.568,Z 451.81,A -85,B 0,C 180,E1 -17396.527,E2 -17396.527} C_VEL
LIN {X 0,Y 294.559,Z 438.159,A -85,B 0,C 180,E1 -17397.025,E2 -17397.025} C_VEL
LIN {X 0,Y 296.267,Z 384.893,A -85,B 0,C 180,E1 -17398.322,E2 -17398.322} C_VEL
LIN {X 0,Y 293.566,Z 366.831,A -85,B 0,C 180,E1 -17399.159,E2 -17399.159} C_VEL
LIN {X 0,Y 290.174,Z 349.172,A -85,B 0,C 180,E1 -17400.097,E2 -17400.097} C_VEL
LIN {X 0,Y 284.269,Z 336.148,A -85,B 0,C 180,E1 -17401.276,E2 -17401.276} C_VEL
LIN {X 0,Y 282.619,Z 332.418,A -85,B 0,C 180,E1 -17401.662,E2 -17401.662} C_VEL
LIN {X 0,Y 280.328,Z 322.42,A -85,B 0,C 180,E1 -17405.212,E2 -17405.212} C_VEL
LIN {X 0,Y 278.089,Z 314.018,A -85,B 0,C 180,E1 -17408.423,E2 -17408.423} C_VEL
LIN {X 0,Y 277.263,Z 310.946,A -85,B 0,C 180,E1 -17409.649,E2 -17409.649} C_VEL
LIN {X 0,Y 277.206,Z 310.955,A -85,B 0,C 180,E1 -17413.197,E2 -17413.197} C_VEL
LIN {X 0,Y 277.212,Z 310.955,A -85,B 0,C 180,E1 -17417.325,E2 -17417.325} C_VEL
LIN {X 0,Y 277.261,Z 310.942,A -85,B 0,C 180,E1 -17421.792,E2 -17421.792} C_VEL
LIN {X 0,Y 277.281,Z 310.941,A -85,B 0,C 180,E1 -17424.341,E2 -17424.341} C_VEL
LIN {X 0,Y 277.24,Z 310.945,A -85,B 0,C 180,E1 -17427.836,E2 -17427.836} C_VEL
LIN {X 0,Y 277.264,Z 310.941,A -85,B 0,C 180,E1 -17431.21,E2 -17431.21} C_VEL
LIN {X 0,Y 277.309,Z 310.939,A -85,B 0,C 180,E1 -17434.479,E2 -17434.479} C_VEL
LIN {X 0,Y 277.287,Z 310.943,A -85,B 0,C 180,E1 -17437.655,E2 -17437.655} C_VEL
LIN {X 0,Y 277.342,Z 310.934,A -85,B 0,C 180,E1 -17440.766,E2 -17440.766} C_VEL
LIN {X 0,Y 277.431,Z 310.927,A -85,B 0,C 180,E1 -17445.326,E2 -17445.326} C_VEL
LIN {X 0,Y 277.503,Z 310.917,A -85,B 0,C 180,E1 -17449.789,E2 -17449.789} C_VEL
LIN {X 0,Y 277.65,Z 310.893,A -85,B 0,C 180,E1 -17452.729,E2 -17452.729} C_VEL
LIN {X 0,Y 277.818,Z 310.878,A -85,B 0,C 180,E1 -17458.551,E2 -17458.551} C_VEL
LIN {X 0,Y 277.818,Z 310.873,A -85,B 0,C 180,E1 -17461.45,E2 -17461.45} C_VEL
LIN {X 0,Y 277.65,Z 310.899,A -85,B 0,C 180,E1 -17467.271,E2 -17467.271} C_VEL
LIN {X 0,Y 277.504,Z 310.912,A -85,B 0,C 180,E1 -17470.212,E2 -17470.212} C_VEL
LIN {X 0,Y 277.432,Z 310.923,A -85,B 0,C 180,E1 -17474.675,E2 -17474.675} C_VEL
LIN {X 0,Y 277.342,Z 310.939,A -85,B 0,C 180,E1 -17479.235,E2 -17479.235} C_VEL
LIN {X 0,Y 277.317,Z 310.939,A -85,B 0,C 180,E1 -17484.171,E2 -17484.171} C_VEL
LIN {X 0,Y 277.321,Z 310.94,A -85,B 0,C 180,E1 -17487.505,E2 -17487.505} C_VEL
LIN {X 0,Y 277.27,Z 310.945,A -85,B 0,C 180,E1 -17490.482,E2 -17490.482} C_VEL
LIN {X 0,Y 277.245,Z 310.948,A -85,B 0,C 180,E1 -17493.897,E2 -17493.897} C_VEL
LIN {X 0,Y 277.261,Z 310.944,A -85,B 0,C 180,E1 -17497.471,E2 -17497.471} C_VEL
LIN {X 0,Y 277.208,Z 310.95,A -85,B 0,C 180,E1 -17501.238,E2 -17501.238} C_VEL
LIN {X 0,Y 277.193,Z 310.955,A -85,B 0,C 180,E1 -17505.229,E2 -17505.229} C_VEL
LIN {X 0,Y 277.211,Z 310.983,A -85,B 0,C 180,E1 -17508.463,E2 -17508.463} C_VEL
LIN {X 0,Y 277.291,Z 311.411,A -85,B 0,C 180,E1 -17508.627,E2 -17508.627} C_VEL
LIN {X 0,Y 278.461,Z 314.173,A -85,B 0,C 180,E1 -17508.891,E2 -17508.891} C_VEL
LIN {X 0,Y 279.871,Z 316.273,A -85,B 0,C 180,E1 -17509.167,E2 -17509.167} C_VEL
LIN {X 0,Y 286.396,Z 327.882,A -85,B 0,C 180,E1 -17510.452,E2 -17510.452} C_VEL
LIN {X 0,Y 293.533,Z 342.332,A -85,B 0,C 180,E1 -17511.819,E2 -17511.819} C_VEL
LIN {X 0,Y 297.362,Z 351.297,A -85,B 0,C 180,E1 -17512.551,E2 -17512.551} C_VEL
LIN {X 0,Y 294.935,Z 417.961,A -85,B 0,C 180,E1 -17514.162,E2 -17514.162} C_VEL
LIN {X 0,Y 294.148,Z 430.884,A -85,B 0,C 180,E1 -17514.743,E2 -17514.743} C_VEL
LIN {X 0,Y 292.797,Z 443.459,A -85,B 0,C 180,E1 -17515.559,E2 -17515.559} C_VEL
LIN {X 0,Y 291.279,Z 454.227,A -85,B 0,C 180,E1 -17516.502,E2 -17516.502} C_VEL
LIN {X 0,Y 289.464,Z 465.002,A -85,B 0,C 180,E1 -17517.715,E2 -17517.715} C_VEL
LIN {X 0,Y 287.427,Z 475.968,A -85,B 0,C 180,E1 -17519.309,E2 -17519.309} C_VEL
LIN {X 0,Y 285.417,Z 484.865,A -85,B 0,C 180,E1 -17520.902,E2 -17520.902} C_VEL
LIN {X 0,Y 283.43,Z 493.004,A -85,B 0,C 180,E1 -17522.696,E2 -17522.696} C_VEL
LIN {X 0,Y 281.421,Z 500.925,A -85,B 0,C 180,E1 -17524.879,E2 -17524.879} C_VEL
LIN {X 0,Y 279.641,Z 507.201,A -85,B 0,C 180,E1 -17527.075,E2 -17527.075} C_VEL
LIN {X 0,Y 278.27,Z 512.154,A -85,B 0,C 180,E1 -17529.294,E2 -17529.294} C_VEL
LIN {X 0,Y 277.169,Z 515.941,A -85,B 0,C 180,E1 -17531.522,E2 -17531.522} C_VEL
LIN {X 0,Y 276.393,Z 518.67,A -85,B 0,C 180,E1 -17533.758,E2 -17533.758} C_VEL
LIN {X 0,Y 275.999,Z 520.041,A -85,B 0,C 180,E1 -17535.384,E2 -17535.384} C_VEL
LIN {X 0,Y 275.451,Z 521.251,A -85,B 0,C 180,E1 -17538.223,E2 -17538.223} C_VEL
LIN {X 0,Y 275.301,Z 520.923,A -85,B 0,C 180,E1 -17541.19,E2 -17541.19} C_VEL
LIN {X 0,Y 275.357,Z 520.181,A -85,B 0,C 180,E1 -17542.669,E2 -17542.669} C_VEL
LIN {X 0,Y 275.533,Z 518.996,A -85,B 0,C 180,E1 -17544.145,E2 -17544.145} C_VEL
LIN {X 0,Y 275.603,Z 517.412,A -85,B 0,C 180,E1 -17545.613,E2 -17545.613} C_VEL
LIN {X 0,Y 275.903,Z 514.237,A -85,B 0,C 180,E1 -17547.811,E2 -17547.811} C_VEL
LIN {X 0,Y 276.42,Z 510.008,A -85,B 0,C 180,E1 -17550.001,E2 -17550.001} C_VEL
LIN {X 0,Y 277.331,Z 503.603,A -85,B 0,C 180,E1 -17552.543,E2 -17552.543} C_VEL
LIN {X 0,Y 278.395,Z 496.595,A -85,B 0,C 180,E1 -17554.707,E2 -17554.707} C_VEL
LIN {X 0,Y 279.745,Z 487.845,A -85,B 0,C 180,E1 -17556.855,E2 -17556.855} C_VEL
LIN {X 0,Y 281.19,Z 477.916,A -85,B 0,C 180,E1 -17558.807,E2 -17558.807} C_VEL
LIN {X 0,Y 282.632,Z 467.754,A -85,B 0,C 180,E1 -17560.387,E2 -17560.387} C_VEL
LIN {X 0,Y 284.004,Z 456.499,A -85,B 0,C 180,E1 -17561.781,E2 -17561.781} C_VEL
LIN {X 0,Y 285.059,Z 444.871,A -85,B 0,C 180,E1 -17562.912,E2 -17562.912} C_VEL
LIN {X 0,Y 286.017,Z 432.862,A -85,B 0,C 180,E1 -17563.772,E2 -17563.772} C_VEL
LIN {X 0,Y 286.69,Z 419.276,A -85,B 0,C 180,E1 -17564.433,E2 -17564.433} C_VEL
LIN {X 0,Y 287.379,Z 394.867,A -85,B 0,C 180,E1 -17565.082,E2 -17565.082} C_VEL
LIN {X 0,Y 288.735,Z 340.944,A -85,B 0,C 180,E1 -17566.398,E2 -17566.398} C_VEL
LIN {X 0,Y 282.579,Z 323.564,A -85,B 0,C 180,E1 -17567.379,E2 -17567.379} C_VEL
LIN {X 0,Y 277.511,Z 311.753,A -85,B 0,C 180,E1 -17568.156,E2 -17568.156} C_VEL
LIN {X 0,Y 277.358,Z 310.938,A -85,B 0,C 180,E1 -17568.228,E2 -17568.228} C_VEL
LIN {X 0,Y 277.266,Z 310.944,A -85,B 0,C 180,E1 -17572.348,E2 -17572.348} C_VEL
LIN {X 0,Y 277.251,Z 310.943,A -85,B 0,C 180,E1 -17575.528,E2 -17575.528} C_VEL
LIN {X 0,Y 277.244,Z 310.949,A -85,B 0,C 180,E1 -17578.794,E2 -17578.794} C_VEL
LIN {X 0,Y 277.245,Z 310.948,A -85,B 0,C 180,E1 -17582.165,E2 -17582.165} C_VEL
LIN {X 0,Y 277.279,Z 310.944,A -85,B 0,C 180,E1 -17585.797,E2 -17585.797} C_VEL
LIN {X 0,Y 277.221,Z 310.952,A -85,B 0,C 180,E1 -17589.331,E2 -17589.331} C_VEL
LIN {X 0,Y 277.196,Z 310.956,A -85,B 0,C 180,E1 -17593.202,E2 -17593.202} C_VEL
LIN {X 0,Y 277.197,Z 310.949,A -85,B 0,C 180,E1 -17597.331,E2 -17597.331} C_VEL
LIN {X 0,Y 277.248,Z 310.948,A -85,B 0,C 180,E1 -17601.798,E2 -17601.798} C_VEL
LIN {X 0,Y 277.284,Z 310.936,A -85,B 0,C 180,E1 -17604.341,E2 -17604.341} C_VEL
LIN {X 0,Y 277.245,Z 310.95,A -85,B 0,C 180,E1 -17607.836,E2 -17607.836} C_VEL
LIN {X 0,Y 277.244,Z 310.949,A -85,B 0,C 180,E1 -17611.207,E2 -17611.207} C_VEL
LIN {X 0,Y 277.244,Z 310.936,A -85,B 0,C 180,E1 -17614.472,E2 -17614.472} C_VEL
LIN {X 0,Y 277.262,Z 310.946,A -85,B 0,C 180,E1 -17617.652,E2 -17617.652} C_VEL
LIN {X 0,Y 277.329,Z 310.936,A -85,B 0,C 180,E1 -17620.765,E2 -17620.765} C_VEL
LIN {X 0,Y 277.325,Z 310.931,A -85,B 0,C 180,E1 -17622.679,E2 -17622.679} C_VEL
LIN {X 0,Y 276.656,Z 311.014,A -85,B 0,C 180,E1 -17623.892,E2 -17623.892} C_VEL
LIN {X 0,Y 273.814,Z 311.367,A -85,B 0,C 180,E1 -17625.868,E2 -17625.868} C_VEL
LIN {X 0,Y 271.431,Z 311.668,A -85,B 0,C 180,E1 -17627.474,E2 -17627.474} C_VEL
LIN {X 0,Y 270.448,Z 311.794,A -85,B 0,C 180,E1 -17628.719,E2 -17628.719} C_VEL
LIN {X 0,Y 270.388,Z 311.8,A -85,B 0,C 180,E1 -17629.14,E2 -17629.14} C_VEL
LIN {X 0,Y 270.567,Z 311.776,A -85,B 0,C 180,E1 -17632.537,E2 -17632.537} C_VEL
LIN {X 0,Y 270.774,Z 311.755,A -85,B 0,C 180,E1 -17638.512,E2 -17638.512} C_VEL
LIN {X 0,Y 270.778,Z 311.753,A -85,B 0,C 180,E1 -17641.487,E2 -17641.487} C_VEL
LIN {X 0,Y 270.566,Z 311.771,A -85,B 0,C 180,E1 -17647.462,E2 -17647.462} C_VEL
LIN {X 0,Y 270.41,Z 311.802,A -85,B 0,C 180,E1 -17650.482,E2 -17650.482} C_VEL
LIN {X 0,Y 270.372,Z 311.805,A -85,B 0,C 180,E1 -17655.066,E2 -17655.066} C_VEL
LIN {X 0,Y 270.228,Z 311.822,A -85,B 0,C 180,E1 -17659.761,E2 -17659.761} C_VEL
LIN {X 0,Y 270.227,Z 311.825,A -85,B 0,C 180,E1 -17664.59,E2 -17664.59} C_VEL
LIN {X 0,Y 270.196,Z 311.826,A -85,B 0,C 180,E1 -17667.917,E2 -17667.917} C_VEL
LIN {X 0,Y 270.172,Z 311.832,A -85,B 0,C 180,E1 -17671.35,E2 -17671.35} C_VEL
LIN {X 0,Y 270.201,Z 311.83,A -85,B 0,C 180,E1 -17674.905,E2 -17674.905} C_VEL
LIN {X 0,Y 270.201,Z 311.828,A -85,B 0,C 180,E1 -17678.71,E2 -17678.71} C_VEL
LIN {X 0,Y 270.15,Z 311.836,A -85,B 0,C 180,E1 -17683.244,E2 -17683.244} C_VEL
LIN {X 0,Y 270.153,Z 311.835,A -85,B 0,C 180,E1 -17687.437,E2 -17687.437} C_VEL
LIN {X 0,Y 270.21,Z 311.829,A -85,B 0,C 180,E1 -17691.373,E2 -17691.373} C_VEL
LIN {X 0,Y 270.256,Z 311.954,A -85,B 0,C 180,E1 -17695.588,E2 -17695.588} C_VEL
LIN {X 0,Y 272.49,Z 321.972,A -85,B 0,C 180,E1 -17698.946,E2 -17698.946} C_VEL
LIN {X 0,Y 274.583,Z 333.253,A -85,B 0,C 180,E1 -17702.527,E2 -17702.527} C_VEL
LIN {X 0,Y 275.748,Z 338.781,A -85,B 0,C 180,E1 -17702.805,E2 -17702.805} C_VEL
LIN {X 0,Y 279.553,Z 367.064,A -85,B 0,C 180,E1 -17703.915,E2 -17703.915} C_VEL
LIN {X 0,Y 281.286,Z 382.422,A -85,B 0,C 180,E1 -17704.475,E2 -17704.475} C_VEL
LIN {X 0,Y 279.846,Z 442.178,A -85,B 0,C 180,E1 -17706.007,E2 -17706.007} C_VEL
LIN {X 0,Y 278.894,Z 455.564,A -85,B 0,C 180,E1 -17706.615,E2 -17706.615} C_VEL
LIN {X 0,Y 277.703,Z 468.337,A -85,B 0,C 180,E1 -17707.493,E2 -17707.493} C_VEL
LIN {X 0,Y 276.305,Z 479.658,A -85,B 0,C 180,E1 -17708.552,E2 -17708.552} C_VEL
LIN {X 0,Y 274.74,Z 491.383,A -85,B 0,C 180,E1 -17709.992,E2 -17709.992} C_VEL
LIN {X 0,Y 273.324,Z 500.84,A -85,B 0,C 180,E1 -17711.445,E2 -17711.445} C_VEL
LIN {X 0,Y 272.051,Z 509.505,A -85,B 0,C 180,E1 -17713.075,E2 -17713.075} C_VEL
LIN {X 0,Y 271.133,Z 516.231,A -85,B 0,C 180,E1 -17714.591,E2 -17714.591} C_VEL
LIN {X 0,Y 269.942,Z 524.436,A -85,B 0,C 180,E1 -17716.831,E2 -17716.831} C_VEL
LIN {X 0,Y 269.177,Z 530.005,A -85,B 0,C 180,E1 -17718.706,E2 -17718.706} C_VEL
LIN {X 0,Y 268.641,Z 535.451,A -85,B 0,C 180,E1 -17720.968,E2 -17720.968} C_VEL
LIN {X 0,Y 268.328,Z 539.688,A -85,B 0,C 180,E1 -17723.23,E2 -17723.23} C_VEL
LIN {X 0,Y 268.249,Z 542.844,A -85,B 0,C 180,E1 -17725.491,E2 -17725.491} C_VEL
LIN {X 0,Y 268.311,Z 544.413,A -85,B 0,C 180,E1 -17726.996,E2 -17726.996} C_VEL
LIN {X 0,Y 268.295,Z 545.529,A -85,B 0,C 180,E1 -17728.498,E2 -17728.498} C_VEL
LIN {X 0,Y 268.328,Z 546.221,A -85,B 0,C 180,E1 -17729.999,E2 -17729.999} C_VEL
LIN {X 0,Y 268.273,Z 546.518,A -85,B 0,C 180,E1 -17731.5,E2 -17731.5} C_VEL
LIN {X 0,Y 268.258,Z 546.427,A -85,B 0,C 180,E1 -17733.003,E2 -17733.003} C_VEL
LIN {X 0,Y 268.231,Z 545.458,A -85,B 0,C 180,E1 -17735.348,E2 -17735.348} C_VEL
LIN {X 0,Y 268.379,Z 543.686,A -85,B 0,C 180,E1 -17737.523,E2 -17737.523} C_VEL
LIN {X 0,Y 268.89,Z 540.933,A -85,B 0,C 180,E1 -17739.781,E2 -17739.781} C_VEL
LIN {X 0,Y 269.642,Z 537.176,A -85,B 0,C 180,E1 -17742.034,E2 -17742.034} C_VEL
LIN {X 0,Y 270.911,Z 532.326,A -85,B 0,C 180,E1 -17744.267,E2 -17744.267} C_VEL
LIN {X 0,Y 272.524,Z 526.235,A -85,B 0,C 180,E1 -17746.479,E2 -17746.479} C_VEL
LIN {X 0,Y 274.429,Z 518.796,A -85,B 0,C 180,E1 -17748.639,E2 -17748.639} C_VEL
LIN {X 0,Y 276.39,Z 511.008,A -85,B 0,C 180,E1 -17750.464,E2 -17750.464} C_VEL
LIN {X 0,Y 278.732,Z 501.687,A -85,B 0,C 180,E1 -17752.222,E2 -17752.222} C_VEL
LIN {X 0,Y 281.031,Z 491.353,A -85,B 0,C 180,E1 -17753.781,E2 -17753.781} C_VEL
LIN {X 0,Y 283.361,Z 479.901,A -85,B 0,C 180,E1 -17755.133,E2 -17755.133} C_VEL
LIN {X 0,Y 285.395,Z 467.922,A -85,B 0,C 180,E1 -17756.213,E2 -17756.213} C_VEL
LIN {X 0,Y 287.092,Z 454.63,A -85,B 0,C 180,E1 -17757.075,E2 -17757.075} C_VEL
LIN {X 0,Y 288.267,Z 441.59,A -85,B 0,C 180,E1 -17757.633,E2 -17757.633} C_VEL
LIN {X 0,Y 290.188,Z 384.861,A -85,B 0,C 180,E1 -17759.062,E2 -17759.062} C_VEL
LIN {X 0,Y 286.25,Z 360.366,A -85,B 0,C 180,E1 -17760.284,E2 -17760.284} C_VEL
LIN {X 0,Y 284.318,Z 351.54,A -85,B 0,C 180,E1 -17760.807,E2 -17760.807} C_VEL
LIN {X 0,Y 278.314,Z 338.422,A -85,B 0,C 180,E1 -17762.056,E2 -17762.056} C_VEL
LIN {X 0,Y 275.365,Z 332.006,A -85,B 0,C 180,E1 -17762.736,E2 -17762.736} C_VEL
LIN {X 0,Y 273.11,Z 322.432,A -85,B 0,C 180,E1 -17766.288,E2 -17766.288} C_VEL
LIN {X 0,Y 270.691,Z 313.601,A -85,B 0,C 180,E1 -17769.838,E2 -17769.838} C_VEL
LIN {X 0,Y 270.172,Z 311.831,A -85,B 0,C 180,E1 -17770.65,E2 -17770.65} C_VEL
LIN {X 0,Y 270.149,Z 311.835,A -85,B 0,C 180,E1 -17774.62,E2 -17774.62} C_VEL
LIN {X 0,Y 270.166,Z 311.826,A -85,B 0,C 180,E1 -17778.971,E2 -17778.971} C_VEL
LIN {X 0,Y 270.214,Z 311.825,A -85,B 0,C 180,E1 -17783.259,E2 -17783.259} C_VEL
LIN {X 0,Y 270.199,Z 311.826,A -85,B 0,C 180,E1 -17786.892,E2 -17786.892} C_VEL
LIN {X 0,Y 270.216,Z 311.824,A -85,B 0,C 180,E1 -17790.385,E2 -17790.385} C_VEL
LIN {X 0,Y 270.259,Z 311.817,A -85,B 0,C 180,E1 -17793.764,E2 -17793.764} C_VEL
LIN {X 0,Y 270.233,Z 311.821,A -85,B 0,C 180,E1 -17797.039,E2 -17797.039} C_VEL
LIN {X 0,Y 270.298,Z 311.806,A -85,B 0,C 180,E1 -17800.244,E2 -17800.244} C_VEL
LIN {X 0,Y 270.399,Z 311.801,A -85,B 0,C 180,E1 -17804.935,E2 -17804.935} C_VEL
LIN {X 0,Y 270.438,Z 311.798,A -85,B 0,C 180,E1 -17809.519,E2 -17809.519} C_VEL
LIN {X 0,Y 270.608,Z 311.769,A -85,B 0,C 180,E1 -17812.539,E2 -17812.539} C_VEL
LIN {X 0,Y 270.784,Z 311.754,A -85,B 0,C 180,E1 -17818.513,E2 -17818.513} C_VEL
LIN {X 0,Y 270.784,Z 311.75,A -85,B 0,C 180,E1 -17821.488,E2 -17821.488} C_VEL
LIN {X 0,Y 270.608,Z 311.775,A -85,B 0,C 180,E1 -17827.462,E2 -17827.462} C_VEL
LIN {X 0,Y 270.439,Z 311.793,A -85,B 0,C 180,E1 -17830.482,E2 -17830.482} C_VEL
LIN {X 0,Y 270.4,Z 311.802,A -85,B 0,C 180,E1 -17835.065,E2 -17835.065} C_VEL
LIN {X 0,Y 270.299,Z 311.814,A -85,B 0,C 180,E1 -17839.756,E2 -17839.756} C_VEL
LIN {X 0,Y 270.272,Z 311.815,A -85,B 0,C 180,E1 -17844.586,E2 -17844.586} C_VEL
LIN {X 0,Y 270.267,Z 311.816,A -85,B 0,C 180,E1 -17847.91,E2 -17847.91} C_VEL
LIN {X 0,Y 270.182,Z 311.825,A -85,B 0,C 180,E1 -17851.349,E2 -17851.349} C_VEL
LIN {X 0,Y 270.199,Z 311.822,A -85,B 0,C 180,E1 -17854.907,E2 -17854.907} C_VEL
LIN {X 0,Y 270.196,Z 311.821,A -85,B 0,C 180,E1 -17858.711,E2 -17858.711} C_VEL
LIN {X 0,Y 270.164,Z 311.829,A -85,B 0,C 180,E1 -17863.25,E2 -17863.25} C_VEL
LIN {X 0,Y 270.165,Z 311.86,A -85,B 0,C 180,E1 -17867.518,E2 -17867.518} C_VEL
LIN {X 0,Y 271.107,Z 314.596,A -85,B 0,C 180,E1 -17867.761,E2 -17867.761} C_VEL
LIN {X 0,Y 272.858,Z 317.11,A -85,B 0,C 180,E1 -17868.122,E2 -17868.122} C_VEL
LIN {X 0,Y 278.975,Z 327.456,A -85,B 0,C 180,E1 -17869.382,E2 -17869.382} C_VEL
LIN {X 0,Y 286.928,Z 343.186,A -85,B 0,C 180,E1 -17870.98,E2 -17870.98} C_VEL
LIN {X 0,Y 291.292,Z 353.249,A -85,B 0,C 180,E1 -17871.848,E2 -17871.848} C_VEL
LIN {X 0,Y 288.883,Z 417.877,A -85,B 0,C 180,E1 -17873.439,E2 -17873.439} C_VEL
LIN {X 0,Y 288.067,Z 430.684,A -85,B 0,C 180,E1 -17874.011,E2 -17874.011} C_VEL
LIN {X 0,Y 286.727,Z 443.19,A -85,B 0,C 180,E1 -17874.831,E2 -17874.831} C_VEL
LIN {X 0,Y 285.176,Z 453.168,A -85,B 0,C 180,E1 -17875.686,E2 -17875.686} C_VEL
LIN {X 0,Y 283.32,Z 464.25,A -85,B 0,C 180,E1 -17876.927,E2 -17876.927} C_VEL
LIN {X 0,Y 281.482,Z 474.379,A -85,B 0,C 180,E1 -17878.378,E2 -17878.378} C_VEL
LIN {X 0,Y 279.509,Z 482.679,A -85,B 0,C 180,E1 -17879.81,E2 -17879.81} C_VEL
LIN {X 0,Y 277.414,Z 491.254,A -85,B 0,C 180,E1 -17881.641,E2 -17881.641} C_VEL
LIN {X 0,Y 275.383,Z 498.841,A -85,B 0,C 180,E1 -17883.644,E2 -17883.644} C_VEL
LIN {X 0,Y 273.522,Z 505.202,A -85,B 0,C 180,E1 -17885.726,E2 -17885.726} C_VEL
LIN {X 0,Y 271.889,Z 510.827,A -85,B 0,C 180,E1 -17888.069,E2 -17888.069} C_VEL
LIN {X 0,Y 270.637,Z 514.901,A -85,B 0,C 180,E1 -17890.271,E2 -17890.271} C_VEL
LIN {X 0,Y 269.956,Z 517.132,A -85,B 0,C 180,E1 -17891.797,E2 -17891.797} C_VEL
LIN {X 0,Y 269.441,Z 518.863,A -85,B 0,C 180,E1 -17893.327,E2 -17893.327} C_VEL
LIN {X 0,Y 268.954,Z 520.419,A -85,B 0,C 180,E1 -17895.207,E2 -17895.207} C_VEL
LIN {X 0,Y 268.394,Z 521.569,A -85,B 0,C 180,E1 -17897.909,E2 -17897.909} C_VEL
LIN {X 0,Y 268.195,Z 521.304,A -85,B 0,C 180,E1 -17900.955,E2 -17900.955} C_VEL
LIN {X 0,Y 268.258,Z 520.592,A -85,B 0,C 180,E1 -17902.474,E2 -17902.474} C_VEL
LIN {X 0,Y 268.447,Z 519.277,A -85,B 0,C 180,E1 -17904.188,E2 -17904.188} C_VEL
LIN {X 0,Y 268.653,Z 515.957,A -85,B 0,C 180,E1 -17907.002,E2 -17907.002} C_VEL
LIN {X 0,Y 269.159,Z 512.153,A -85,B 0,C 180,E1 -17909.253,E2 -17909.253} C_VEL
LIN {X 0,Y 269.799,Z 507.242,A -85,B 0,C 180,E1 -17911.494,E2 -17911.494} C_VEL
LIN {X 0,Y 270.771,Z 501.063,A -85,B 0,C 180,E1 -17913.721,E2 -17913.721} C_VEL
LIN {X 0,Y 271.971,Z 493.361,A -85,B 0,C 180,E1 -17915.934,E2 -17915.934} C_VEL
LIN {X 0,Y 273.505,Z 483.717,A -85,B 0,C 180,E1 -17918.126,E2 -17918.126} C_VEL
LIN {X 0,Y 274.986,Z 473.754,A -85,B 0,C 180,E1 -17919.935,E2 -17919.935} C_VEL
LIN {X 0,Y 276.537,Z 462.459,A -85,B 0,C 180,E1 -17921.546,E2 -17921.546} C_VEL
LIN {X 0,Y 277.824,Z 451.405,A -85,B 0,C 180,E1 -17922.789,E2 -17922.789} C_VEL
LIN {X 0,Y 278.854,Z 439.142,A -85,B 0,C 180,E1 -17923.854,E2 -17923.854} C_VEL
LIN {X 0,Y 279.757,Z 426.113,A -85,B 0,C 180,E1 -17924.64,E2 -17924.64} C_VEL
LIN {X 0,Y 280.255,Z 412.774,A -85,B 0,C 180,E1 -17925.151,E2 -17925.151} C_VEL
LIN {X 0,Y 282.175,Z 342.321,A -85,B 0,C 180,E1 -17926.904,E2 -17926.904} C_VEL
LIN {X 0,Y 275.6,Z 324.225,A -85,B 0,C 180,E1 -17927.982,E2 -17927.982} C_VEL
LIN {X 0,Y 270.403,Z 312.401,A -85,B 0,C 180,E1 -17928.805,E2 -17928.805} C_VEL
LIN {X 0,Y 270.304,Z 311.816,A -85,B 0,C 180,E1 -17928.878,E2 -17928.878} C_VEL
LIN {X 0,Y 270.205,Z 311.825,A -85,B 0,C 180,E1 -17932.965,E2 -17932.965} C_VEL
LIN {X 0,Y 270.207,Z 311.82,A -85,B 0,C 180,E1 -17936.243,E2 -17936.243} C_VEL
LIN {X 0,Y 270.188,Z 311.827,A -85,B 0,C 180,E1 -17939.619,E2 -17939.619} C_VEL
LIN {X 0,Y 270.22,Z 311.824,A -85,B 0,C 180,E1 -17943.666,E2 -17943.666} C_VEL
LIN {X 0,Y 270.214,Z 311.826,A -85,B 0,C 180,E1 -17946.743,E2 -17946.743} C_VEL
LIN {X 0,Y 270.153,Z 311.829,A -85,B 0,C 180,E1 -17950.571,E2 -17950.571} C_VEL
LIN {X 0,Y 270.133,Z 311.833,A -85,B 0,C 180,E1 -17954.625,E2 -17954.625} C_VEL
LIN {X 0,Y 270.156,Z 311.825,A -85,B 0,C 180,E1 -17957.438,E2 -17957.438} C_VEL
LIN {X 0,Y 270.173,Z 311.832,A -85,B 0,C 180,E1 -17961.368,E2 -17961.368} C_VEL
LIN {X 0,Y 270.204,Z 311.819,A -85,B 0,C 180,E1 -17965.094,E2 -17965.094} C_VEL
LIN {X 0,Y 270.189,Z 311.827,A -85,B 0,C 180,E1 -17969.136,E2 -17969.136} C_VEL
LIN {X 0,Y 270.227,Z 311.819,A -85,B 0,C 180,E1 -17972.163,E2 -17972.163} C_VEL
LIN {X 0,Y 270.222,Z 311.813,A -85,B 0,C 180,E1 -17975.547,E2 -17975.547} C_VEL
LIN {X 0,Y 270.266,Z 311.818,A -85,B 0,C 180,E1 -17980.241,E2 -17980.241} C_VEL
LIN {X 0,Y 270.382,Z 311.789,A -85,B 0,C 180,E1 -17984.934,E2 -17984.934} C_VEL
LIN {X 0,Y 270.388,Z 311.8,A -85,B 0,C 180,E1 -17989.14,E2 -17989.14} C_VEL
LIN {X 0,Y 269.757,Z 311.883,A -85,B 0,C 180,E1 -17990.385,E2 -17990.385} C_VEL
LIN {X 0,Y 266.866,Z 312.238,A -85,B 0,C 180,E1 -17992.411,E2 -17992.411} C_VEL
LIN {X 0,Y 264.42,Z 312.537,A -85,B 0,C 180,E1 -17994.06,E2 -17994.06} C_VEL
LIN {X 0,Y 263.421,Z 312.655,A -85,B 0,C 180,E1 -17995.34,E2 -17995.34} C_VEL
LIN {X 0,Y 263.369,Z 312.661,A -85,B 0,C 180,E1 -17995.773,E2 -17995.773} C_VEL
LIN {X 0,Y 263.738,Z 312.63,A -85,B 0,C 180,E1 -17998.473,E2 -17998.473} C_VEL
LIN {X 0,Y 263.741,Z 312.63,A -85,B 0,C 180,E1 -18001.527,E2 -18001.527} C_VEL
LIN {X 0,Y 263.53,Z 312.647,A -85,B 0,C 180,E1 -18007.663,E2 -18007.663} C_VEL
LIN {X 0,Y 263.35,Z 312.682,A -85,B 0,C 180,E1 -18010.766,E2 -18010.766} C_VEL
LIN {X 0,Y 263.314,Z 312.683,A -85,B 0,C 180,E1 -18015.48,E2 -18015.48} C_VEL
LIN {X 0,Y 263.213,Z 312.697,A -85,B 0,C 180,E1 -18020.31,E2 -18020.31} C_VEL
LIN {X 0,Y 263.17,Z 312.703,A -85,B 0,C 180,E1 -18025.295,E2 -18025.295} C_VEL
LIN {X 0,Y 263.125,Z 312.711,A -85,B 0,C 180,E1 -18028.736,E2 -18028.736} C_VEL
LIN {X 0,Y 263.129,Z 312.708,A -85,B 0,C 180,E1 -18032.288,E2 -18032.288} C_VEL
LIN {X 0,Y 263.179,Z 312.704,A -85,B 0,C 180,E1 -18036.76,E2 -18036.76} C_VEL
LIN {X 0,Y 263.094,Z 312.712,A -85,B 0,C 180,E1 -18039.874,E2 -18039.874} C_VEL
LIN {X 0,Y 263.079,Z 312.713,A -85,B 0,C 180,E1 -18043.993,E2 -18043.993} C_VEL
LIN {X 0,Y 263.083,Z 312.712,A -85,B 0,C 180,E1 -18048.417,E2 -18048.417} C_VEL
LIN {X 0,Y 263.16,Z 312.706,A -85,B 0,C 180,E1 -18052.102,E2 -18052.102} C_VEL
LIN {X 0,Y 263.211,Z 312.874,A -85,B 0,C 180,E1 -18055.093,E2 -18055.093} C_VEL
LIN {X 0,Y 265.696,Z 324.051,A -85,B 0,C 180,E1 -18058.948,E2 -18058.948} C_VEL
LIN {X 0,Y 267.359,Z 332.918,A -85,B 0,C 180,E1 -18061.848,E2 -18061.848} C_VEL
LIN {X 0,Y 269.205,Z 339.401,A -85,B 0,C 180,E1 -18062.222,E2 -18062.222} C_VEL
LIN {X 0,Y 272.81,Z 366.617,A -85,B 0,C 180,E1 -18063.323,E2 -18063.323} C_VEL
LIN {X 0,Y 274.698,Z 384.211,A -85,B 0,C 180,E1 -18063.978,E2 -18063.978} C_VEL
LIN {X 0,Y 273.215,Z 442.022,A -85,B 0,C 180,E1 -18065.496,E2 -18065.496} C_VEL
LIN {X 0,Y 272.236,Z 455.236,A -85,B 0,C 180,E1 -18066.109,E2 -18066.109} C_VEL
LIN {X 0,Y 271.002,Z 468.008,A -85,B 0,C 180,E1 -18067.006,E2 -18067.006} C_VEL
LIN {X 0,Y 269.46,Z 480.129,A -85,B 0,C 180,E1 -18068.181,E2 -18068.181} C_VEL
LIN {X 0,Y 267.831,Z 491.705,A -85,B 0,C 180,E1 -18069.653,E2 -18069.653} C_VEL
LIN {X 0,Y 266.249,Z 502.136,A -85,B 0,C 180,E1 -18071.333,E2 -18071.333} C_VEL
LIN {X 0,Y 264.992,Z 510.663,A -85,B 0,C 180,E1 -18073.037,E2 -18073.037} C_VEL
LIN {X 0,Y 263.746,Z 518.51,A -85,B 0,C 180,E1 -18074.94,E2 -18074.94} C_VEL
LIN {X 0,Y 262.582,Z 526.171,A -85,B 0,C 180,E1 -18077.242,E2 -18077.242} C_VEL
LIN {X 0,Y 261.721,Z 533.249,A -85,B 0,C 180,E1 -18079.947,E2 -18079.947} C_VEL
LIN {X 0,Y 261.346,Z 537.927,A -85,B 0,C 180,E1 -18082.272,E2 -18082.272} C_VEL
LIN {X 0,Y 261.178,Z 541.535,A -85,B 0,C 180,E1 -18084.64,E2 -18084.64} C_VEL
LIN {X 0,Y 261.217,Z 543.994,A -85,B 0,C 180,E1 -18086.914,E2 -18086.914} C_VEL
LIN {X 0,Y 261.219,Z 545.15,A -85,B 0,C 180,E1 -18088.457,E2 -18088.457} C_VEL
LIN {X 0,Y 261.248,Z 545.862,A -85,B 0,C 180,E1 -18089.999,E2 -18089.999} C_VEL
LIN {X 0,Y 261.197,Z 546.178,A -85,B 0,C 180,E1 -18091.541,E2 -18091.541} C_VEL
LIN {X 0,Y 261.165,Z 546.106,A -85,B 0,C 180,E1 -18093.084,E2 -18093.084} C_VEL
LIN {X 0,Y 261.131,Z 545.308,A -85,B 0,C 180,E1 -18095.248,E2 -18095.248} C_VEL
LIN {X 0,Y 261.321,Z 543.443,A -85,B 0,C 180,E1 -18097.727,E2 -18097.727} C_VEL
LIN {X 0,Y 261.849,Z 540.733,A -85,B 0,C 180,E1 -18100.046,E2 -18100.046} C_VEL
LIN {X 0,Y 262.657,Z 537.021,A -85,B 0,C 180,E1 -18102.359,E2 -18102.359} C_VEL
LIN {X 0,Y 264.003,Z 532.219,A -85,B 0,C 180,E1 -18104.648,E2 -18104.648} C_VEL
LIN {X 0,Y 265.688,Z 526.181,A -85,B 0,C 180,E1 -18106.915,E2 -18106.915} C_VEL
LIN {X 0,Y 267.533,Z 519.383,A -85,B 0,C 180,E1 -18108.967,E2 -18108.967} C_VEL
LIN {X 0,Y 269.749,Z 511.081,A -85,B 0,C 180,E1 -18110.991,E2 -18110.991} C_VEL
LIN {X 0,Y 272.186,Z 501.878,A -85,B 0,C 180,E1 -18112.786,E2 -18112.786} C_VEL
LIN {X 0,Y 274.561,Z 491.663,A -85,B 0,C 180,E1 -18114.377,E2 -18114.377} C_VEL
LIN {X 0,Y 276.985,Z 480.355,A -85,B 0,C 180,E1 -18115.754,E2 -18115.754} C_VEL
LIN {X 0,Y 279.079,Z 468.632,A -85,B 0,C 180,E1 -18116.853,E2 -18116.853} C_VEL
LIN {X 0,Y 280.749,Z 456.565,A -85,B 0,C 180,E1 -18117.688,E2 -18117.688} C_VEL
LIN {X 0,Y 282.02,Z 443.445,A -85,B 0,C 180,E1 -18118.303,E2 -18118.303} C_VEL
LIN {X 0,Y 282.971,Z 421.305,A -85,B 0,C 180,E1 -18118.909,E2 -18118.909} C_VEL
LIN {X 0,Y 284.163,Z 385.711,A -85,B 0,C 180,E1 -18119.808,E2 -18119.808} C_VEL
LIN {X 0,Y 280.442,Z 362.249,A -85,B 0,C 180,E1 -18121.018,E2 -18121.018} C_VEL
LIN {X 0,Y 278.641,Z 354.212,A -85,B 0,C 180,E1 -18121.52,E2 -18121.52} C_VEL
LIN {X 0,Y 272.317,Z 340.344,A -85,B 0,C 180,E1 -18122.896,E2 -18122.896} C_VEL
LIN {X 0,Y 268.073,Z 331.557,A -85,B 0,C 180,E1 -18123.9,E2 -18123.9} C_VEL
LIN {X 0,Y 265.826,Z 322.26,A -85,B 0,C 180,E1 -18127.519,E2 -18127.519} C_VEL
LIN {X 0,Y 263.752,Z 314.901,A -85,B 0,C 180,E1 -18130.621,E2 -18130.621} C_VEL
LIN {X 0,Y 263.126,Z 312.705,A -85,B 0,C 180,E1 -18131.675,E2 -18131.675} C_VEL
LIN {X 0,Y 263.1,Z 312.708,A -85,B 0,C 180,E1 -18136.011,E2 -18136.011} C_VEL
LIN {X 0,Y 263.102,Z 312.71,A -85,B 0,C 180,E1 -18140.127,E2 -18140.127} C_VEL
LIN {X 0,Y 263.16,Z 312.703,A -85,B 0,C 180,E1 -18144.018,E2 -18144.018} C_VEL
LIN {X 0,Y 263.129,Z 312.703,A -85,B 0,C 180,E1 -18147.711,E2 -18147.711} C_VEL
LIN {X 0,Y 263.194,Z 312.691,A -85,B 0,C 180,E1 -18151.784,E2 -18151.784} C_VEL
LIN {X 0,Y 263.222,Z 312.687,A -85,B 0,C 180,E1 -18155.2,E2 -18155.2} C_VEL
LIN {X 0,Y 263.261,Z 312.681,A -85,B 0,C 180,E1 -18159.693,E2 -18159.693} C_VEL
LIN {X 0,Y 263.347,Z 312.675,A -85,B 0,C 180,E1 -18164.522,E2 -18164.522} C_VEL
LIN {X 0,Y 263.371,Z 312.678,A -85,B 0,C 180,E1 -18169.235,E2 -18169.235} C_VEL
LIN {X 0,Y 263.569,Z 312.644,A -85,B 0,C 180,E1 -18172.339,E2 -18172.339} C_VEL
LIN {X 0,Y 263.749,Z 312.631,A -85,B 0,C 180,E1 -18178.473,E2 -18178.473} C_VEL
LIN {X 0,Y 263.748,Z 312.626,A -85,B 0,C 180,E1 -18181.527,E2 -18181.527} C_VEL
LIN {X 0,Y 263.57,Z 312.65,A -85,B 0,C 180,E1 -18187.662,E2 -18187.662} C_VEL
LIN {X 0,Y 263.371,Z 312.675,A -85,B 0,C 180,E1 -18190.766,E2 -18190.766} C_VEL
LIN {X 0,Y 263.348,Z 312.681,A -85,B 0,C 180,E1 -18195.479,E2 -18195.479} C_VEL
LIN {X 0,Y 263.261,Z 312.691,A -85,B 0,C 180,E1 -18200.307,E2 -18200.307} C_VEL
LIN {X 0,Y 263.206,Z 312.692,A -85,B 0,C 180,E1 -18205.292,E2 -18205.292} C_VEL
LIN {X 0,Y 263.163,Z 312.697,A -85,B 0,C 180,E1 -18208.732,E2 -18208.732} C_VEL
LIN {X 0,Y 263.131,Z 312.699,A -85,B 0,C 180,E1 -18212.289,E2 -18212.289} C_VEL
LIN {X 0,Y 263.179,Z 312.7,A -85,B 0,C 180,E1 -18216.764,E2 -18216.764} C_VEL
LIN {X 0,Y 263.123,Z 312.705,A -85,B 0,C 180,E1 -18221.595,E2 -18221.595} C_VEL
LIN {X 0,Y 263.097,Z 312.71,A -85,B 0,C 180,E1 -18226.012,E2 -18226.012} C_VEL
LIN {X 0,Y 263.119,Z 312.796,A -85,B 0,C 180,E1 -18226.36,E2 -18226.36} C_VEL
LIN {X 0,Y 264.09,Z 315.551,A -85,B 0,C 180,E1 -18226.623,E2 -18226.623} C_VEL
LIN {X 0,Y 265.799,Z 317.854,A -85,B 0,C 180,E1 -18226.993,E2 -18226.993} C_VEL
LIN {X 0,Y 273.045,Z 329.836,A -85,B 0,C 180,E1 -18228.562,E2 -18228.562} C_VEL
LIN {X 0,Y 280.787,Z 344.963,A -85,B 0,C 180,E1 -18230.184,E2 -18230.184} C_VEL
LIN {X 0,Y 285.311,Z 355.286,A -85,B 0,C 180,E1 -18231.122,E2 -18231.122} C_VEL
LIN {X 0,Y 282.796,Z 418.841,A -85,B 0,C 180,E1 -18232.717,E2 -18232.717} C_VEL
LIN {X 0,Y 281.95,Z 431.584,A -85,B 0,C 180,E1 -18233.313,E2 -18233.313} C_VEL
LIN {X 0,Y 280.525,Z 444.071,A -85,B 0,C 180,E1 -18234.155,E2 -18234.155} C_VEL
LIN {X 0,Y 278.915,Z 453.926,A -85,B 0,C 180,E1 -18235.024,E2 -18235.024} C_VEL
LIN {X 0,Y 277.012,Z 464.857,A -85,B 0,C 180,E1 -18236.281,E2 -18236.281} C_VEL
LIN {X 0,Y 275.059,Z 474.971,A -85,B 0,C 180,E1 -18237.767,E2 -18237.767} C_VEL
LIN {X 0,Y 272.777,Z 484.144,A -85,B 0,C 180,E1 -18239.414,E2 -18239.414} C_VEL
LIN {X 0,Y 270.595,Z 492.516,A -85,B 0,C 180,E1 -18241.284,E2 -18241.284} C_VEL
LIN {X 0,Y 268.316,Z 500.67,A -85,B 0,C 180,E1 -18243.56,E2 -18243.56} C_VEL
LIN {X 0,Y 266.288,Z 507.165,A -85,B 0,C 180,E1 -18245.854,E2 -18245.854} C_VEL
LIN {X 0,Y 264.58,Z 512.655,A -85,B 0,C 180,E1 -18248.39,E2 -18248.39} C_VEL
LIN {X 0,Y 263.054,Z 517.263,A -85,B 0,C 180,E1 -18251.302,E2 -18251.302} C_VEL
LIN {X 0,Y 262.491,Z 519.059,A -85,B 0,C 180,E1 -18252.872,E2 -18252.872} C_VEL
LIN {X 0,Y 261.911,Z 520.8,A -85,B 0,C 180,E1 -18255.021,E2 -18255.021} C_VEL
LIN {X 0,Y 261.355,Z 521.872,A -85,B 0,C 180,E1 -18257.578,E2 -18257.578} C_VEL
LIN {X 0,Y 261.148,Z 521.981,A -85,B 0,C 180,E1 -18259.143,E2 -18259.143} C_VEL
LIN {X 0,Y 261.158,Z 521.002,A -85,B 0,C 180,E1 -18262.268,E2 -18262.268} C_VEL
LIN {X 0,Y 261.355,Z 519.541,A -85,B 0,C 180,E1 -18264.249,E2 -18264.249} C_VEL
LIN {X 0,Y 261.56,Z 516.489,A -85,B 0,C 180,E1 -18266.92,E2 -18266.92} C_VEL
LIN {X 0,Y 262.073,Z 512.753,A -85,B 0,C 180,E1 -18269.233,E2 -18269.233} C_VEL
LIN {X 0,Y 262.731,Z 507.914,A -85,B 0,C 180,E1 -18271.534,E2 -18271.534} C_VEL
LIN {X 0,Y 263.717,Z 501.814,A -85,B 0,C 180,E1 -18273.821,E2 -18273.821} C_VEL
LIN {X 0,Y 264.941,Z 494.243,A -85,B 0,C 180,E1 -18276.092,E2 -18276.092} C_VEL
LIN {X 0,Y 266.529,Z 484.718,A -85,B 0,C 180,E1 -18278.34,E2 -18278.34} C_VEL
LIN {X 0,Y 268.039,Z 474.904,A -85,B 0,C 180,E1 -18280.195,E2 -18280.195} C_VEL
LIN {X 0,Y 269.619,Z 463.869,A -85,B 0,C 180,E1 -18281.846,E2 -18281.846} C_VEL
LIN {X 0,Y 270.987,Z 453.061,A -85,B 0,C 180,E1 -18283.117,E2 -18283.117} C_VEL
LIN {X 0,Y 272.017,Z 441.209,A -85,B 0,C 180,E1 -18284.209,E2 -18284.209} C_VEL
LIN {X 0,Y 273.025,Z 428.23,A -85,B 0,C 180,E1 -18285.061,E2 -18285.061} C_VEL
LIN {X 0,Y 273.573,Z 415.381,A -85,B 0,C 180,E1 -18285.602,E2 -18285.602} C_VEL
LIN {X 0,Y 275.601,Z 343.894,A -85,B 0,C 180,E1 -18287.432,E2 -18287.432} C_VEL
LIN {X 0,Y 269.807,Z 327.773,A -85,B 0,C 180,E1 -18288.421,E2 -18288.421} C_VEL
LIN {X 0,Y 264.032,Z 315.186,A -85,B 0,C 180,E1 -18289.354,E2 -18289.354} C_VEL
LIN {X 0,Y 263.24,Z 312.694,A -85,B 0,C 180,E1 -18289.544,E2 -18289.544} C_VEL
LIN {X 0,Y 263.194,Z 312.69,A -85,B 0,C 180,E1 -18294.783,E2 -18294.783} C_VEL
LIN {X 0,Y 263.138,Z 312.706,A -85,B 0,C 180,E1 -18298.736,E2 -18298.736} C_VEL
LIN {X 0,Y 263.133,Z 312.706,A -85,B 0,C 180,E1 -18302.289,E2 -18302.289} C_VEL
LIN {X 0,Y 263.181,Z 312.702,A -85,B 0,C 180,E1 -18306.762,E2 -18306.762} C_VEL
LIN {X 0,Y 263.096,Z 312.707,A -85,B 0,C 180,E1 -18309.875,E2 -18309.875} C_VEL
LIN {X 0,Y 263.081,Z 312.712,A -85,B 0,C 180,E1 -18313.994,E2 -18313.994} C_VEL
LIN {X 0,Y 263.078,Z 312.706,A -85,B 0,C 180,E1 -18318.419,E2 -18318.419} C_VEL
LIN {X 0,Y 263.181,Z 312.7,A -85,B 0,C 180,E1 -18323.239,E2 -18323.239} C_VEL
LIN {X 0,Y 263.133,Z 312.705,A -85,B 0,C 180,E1 -18327.711,E2 -18327.711} C_VEL
LIN {X 0,Y 263.152,Z 312.703,A -85,B 0,C 180,E1 -18331.805,E2 -18331.805} C_VEL
LIN {X 0,Y 263.142,Z 312.701,A -85,B 0,C 180,E1 -18336.382,E2 -18336.382} C_VEL
LIN {X 0,Y 263.243,Z 312.695,A -85,B 0,C 180,E1 -18339.691,E2 -18339.691} C_VEL
LIN {X 0,Y 263.329,Z 312.668,A -85,B 0,C 180,E1 -18344.52,E2 -18344.52} C_VEL
LIN {X 0,Y 263.354,Z 312.677,A -85,B 0,C 180,E1 -18349.233,E2 -18349.233} C_VEL
LIN {X 0,Y 263.531,Z 312.653,A -85,B 0,C 180,E1 -18352.337,E2 -18352.337} C_VEL
LIN {X 0,Y 263.369,Z 312.661,A -85,B 0,C 180,E1 -18355.773,E2 -18355.773} C_VEL
LIN {X 0,Y 262.823,Z 312.737,A -85,B 0,C 180,E1 -18357.053,E2 -18357.053} C_VEL
LIN {X 0,Y 260.147,Z 313.076,A -85,B 0,C 180,E1 -18359.143,E2 -18359.143} C_VEL
LIN {X 0,Y 256.919,Z 313.48,A -85,B 0,C 180,E1 -18361.714,E2 -18361.714} C_VEL
LIN {X 0,Y 256.517,Z 313.525,A -85,B 0,C 180,E1 -18362.602,E2 -18362.602} C_VEL
LIN {X 0,Y 256.458,Z 313.524,A -85,B 0,C 180,E1 -18366.293,E2 -18366.293} C_VEL
LIN {X 0,Y 256.431,Z 313.538,A -85,B 0,C 180,E1 -18369.464,E2 -18369.464} C_VEL
LIN {X 0,Y 256.236,Z 313.565,A -85,B 0,C 180,E1 -18374.291,E2 -18374.291} C_VEL
LIN {X 0,Y 256.167,Z 313.573,A -85,B 0,C 180,E1 -18377.565,E2 -18377.565} C_VEL
LIN {X 0,Y 256.126,Z 313.581,A -85,B 0,C 180,E1 -18381.098,E2 -18381.098} C_VEL
LIN {X 0,Y 256.136,Z 313.581,A -85,B 0,C 180,E1 -18385.111,E2 -18385.111} C_VEL
LIN {X 0,Y 256.046,Z 313.59,A -85,B 0,C 180,E1 -18389.608,E2 -18389.608} C_VEL
LIN {X 0,Y 256.068,Z 313.59,A -85,B 0,C 180,E1 -18393.292,E2 -18393.292} C_VEL
LIN {X 0,Y 256.113,Z 313.585,A -85,B 0,C 180,E1 -18397.269,E2 -18397.269} C_VEL
LIN {X 0,Y 256.021,Z 313.596,A -85,B 0,C 180,E1 -18401.21,E2 -18401.21} C_VEL
LIN {X 0,Y 256.02,Z 313.594,A -85,B 0,C 180,E1 -18405.539,E2 -18405.539} C_VEL
LIN {X 0,Y 256.021,Z 313.592,A -85,B 0,C 180,E1 -18408.789,E2 -18408.789} C_VEL
LIN {X 0,Y 256.131,Z 313.582,A -85,B 0,C 180,E1 -18412.866,E2 -18412.866} C_VEL
LIN {X 0,Y 256.151,Z 313.631,A -85,B 0,C 180,E1 -18414.516,E2 -18414.516} C_VEL
LIN {X 0,Y 258.637,Z 324.937,A -85,B 0,C 180,E1 -18418.537,E2 -18418.537} C_VEL
LIN {X 0,Y 260.128,Z 332.608,A -85,B 0,C 180,E1 -18421.132,E2 -18421.132} C_VEL
LIN {X 0,Y 262.782,Z 340.605,A -85,B 0,C 180,E1 -18421.637,E2 -18421.637} C_VEL
LIN {X 0,Y 266.524,Z 369.317,A -85,B 0,C 180,E1 -18422.832,E2 -18422.832} C_VEL
LIN {X 0,Y 268.135,Z 385.241,A -85,B 0,C 180,E1 -18423.435,E2 -18423.435} C_VEL
LIN {X 0,Y 266.567,Z 442.304,A -85,B 0,C 180,E1 -18424.975,E2 -18424.975} C_VEL
LIN {X 0,Y 265.526,Z 455.672,A -85,B 0,C 180,E1 -18425.622,E2 -18425.622} C_VEL
LIN {X 0,Y 264.306,Z 467.675,A -85,B 0,C 180,E1 -18426.492,E2 -18426.492} C_VEL
LIN {X 0,Y 262.858,Z 479.004,A -85,B 0,C 180,E1 -18427.603,E2 -18427.603} C_VEL
LIN {X 0,Y 261.165,Z 490.726,A -85,B 0,C 180,E1 -18429.11,E2 -18429.11} C_VEL
LIN {X 0,Y 259.456,Z 501.264,A -85,B 0,C 180,E1 -18430.825,E2 -18430.825} C_VEL
LIN {X 0,Y 258.069,Z 509.881,A -85,B 0,C 180,E1 -18432.568,E2 -18432.568} C_VEL
LIN {X 0,Y 257.121,Z 516.328,A -85,B 0,C 180,E1 -18434.136,E2 -18434.136} C_VEL
LIN {X 0,Y 255.846,Z 524.404,A -85,B 0,C 180,E1 -18436.496,E2 -18436.496} C_VEL
LIN {X 0,Y 254.927,Z 530.854,A -85,B 0,C 180,E1 -18438.872,E2 -18438.872} C_VEL
LIN {X 0,Y 254.407,Z 535.974,A -85,B 0,C 180,E1 -18441.26,E2 -18441.26} C_VEL
LIN {X 0,Y 254.151,Z 539.933,A -85,B 0,C 180,E1 -18443.648,E2 -18443.648} C_VEL
LIN {X 0,Y 254.069,Z 541.962,A -85,B 0,C 180,E1 -18445.239,E2 -18445.239} C_VEL
LIN {X 0,Y 254.125,Z 543.572,A -85,B 0,C 180,E1 -18446.828,E2 -18446.828} C_VEL
LIN {X 0,Y 254.145,Z 544.763,A -85,B 0,C 180,E1 -18448.414,E2 -18448.414} C_VEL
LIN {X 0,Y 254.17,Z 545.503,A -85,B 0,C 180,E1 -18449.999,E2 -18449.999} C_VEL
LIN {X 0,Y 254.122,Z 545.839,A -85,B 0,C 180,E1 -18451.584,E2 -18451.584} C_VEL
LIN {X 0,Y 254.075,Z 545.785,A -85,B 0,C 180,E1 -18453.17,E2 -18453.17} C_VEL
LIN {X 0,Y 254.053,Z 545.13,A -85,B 0,C 180,E1 -18455.198,E2 -18455.198} C_VEL
LIN {X 0,Y 254.261,Z 543.202,A -85,B 0,C 180,E1 -18457.943,E2 -18457.943} C_VEL
LIN {X 0,Y 254.817,Z 540.532,A -85,B 0,C 180,E1 -18460.326,E2 -18460.326} C_VEL
LIN {X 0,Y 255.687,Z 536.866,A -85,B 0,C 180,E1 -18462.702,E2 -18462.702} C_VEL
LIN {X 0,Y 257.12,Z 532.112,A -85,B 0,C 180,E1 -18465.049,E2 -18465.049} C_VEL
LIN {X 0,Y 258.881,Z 526.127,A -85,B 0,C 180,E1 -18467.374,E2 -18467.374} C_VEL
LIN {X 0,Y 260.937,Z 518.862,A -85,B 0,C 180,E1 -18469.624,E2 -18469.624} C_VEL
LIN {X 0,Y 263.123,Z 511.155,A -85,B 0,C 180,E1 -18471.546,E2 -18471.546} C_VEL
LIN {X 0,Y 265.658,Z 502.045,A -85,B 0,C 180,E1 -18473.379,E2 -18473.379} C_VEL
LIN {X 0,Y 268.129,Z 491.981,A -85,B 0,C 180,E1 -18475.001,E2 -18475.001} C_VEL
LIN {X 0,Y 270.643,Z 480.822,A -85,B 0,C 180,E1 -18476.403,E2 -18476.403} C_VEL
LIN {X 0,Y 272.624,Z 470.298,A -85,B 0,C 180,E1 -18477.438,E2 -18477.438} C_VEL
LIN {X 0,Y 274.518,Z 457.668,A -85,B 0,C 180,E1 -18478.373,E2 -18478.373} C_VEL
LIN {X 0,Y 275.932,Z 444.31,A -85,B 0,C 180,E1 -18479.037,E2 -18479.037} C_VEL
LIN {X 0,Y 276.776,Z 426.777,A -85,B 0,C 180,E1 -18479.555,E2 -18479.555} C_VEL
LIN {X 0,Y 278.213,Z 386.924,A -85,B 0,C 180,E1 -18480.574,E2 -18480.574} C_VEL
LIN {X 0,Y 274.675,Z 363.995,A -85,B 0,C 180,E1 -18481.79,E2 -18481.79} C_VEL
LIN {X 0,Y 273.122,Z 357.146,A -85,B 0,C 180,E1 -18482.236,E2 -18482.236} C_VEL
LIN {X 0,Y 267.076,Z 343.922,A -85,B 0,C 180,E1 -18483.607,E2 -18483.607} C_VEL
LIN {X 0,Y 262.228,Z 334.341,A -85,B 0,C 180,E1 -18484.737,E2 -18484.737} C_VEL
LIN {X 0,Y 260.785,Z 331.084,A -85,B 0,C 180,E1 -18485.158,E2 -18485.158} C_VEL
LIN {X 0,Y 258.599,Z 322.48,A -85,B 0,C 180,E1 -18488.686,E2 -18488.686} C_VEL
LIN {X 0,Y 256.798,Z 316.216,A -85,B 0,C 180,E1 -18491.454,E2 -18491.454} C_VEL
LIN {X 0,Y 256.065,Z 313.59,A -85,B 0,C 180,E1 -18492.684,E2 -18492.684} C_VEL
LIN {X 0,Y 256.045,Z 313.587,A -85,B 0,C 180,E1 -18496.67,E2 -18496.67} C_VEL
LIN {X 0,Y 256.068,Z 313.587,A -85,B 0,C 180,E1 -18500.858,E2 -18500.858} C_VEL
LIN {X 0,Y 256.127,Z 313.576,A -85,B 0,C 180,E1 -18502.867,E2 -18502.867} C_VEL
LIN {X 0,Y 256.064,Z 313.588,A -85,B 0,C 180,E1 -18506.707,E2 -18506.707} C_VEL
LIN {X 0,Y 256.107,Z 313.582,A -85,B 0,C 180,E1 -18510.4,E2 -18510.4} C_VEL
LIN {X 0,Y 256.185,Z 313.566,A -85,B 0,C 180,E1 -18514.861,E2 -18514.861} C_VEL
LIN {X 0,Y 256.166,Z 313.566,A -85,B 0,C 180,E1 -18519.105,E2 -18519.105} C_VEL
LIN {X 0,Y 256.296,Z 313.551,A -85,B 0,C 180,E1 -18524.085,E2 -18524.085} C_VEL
LIN {X 0,Y 256.306,Z 313.554,A -85,B 0,C 180,E1 -18528.934,E2 -18528.934} C_VEL
LIN {X 0,Y 256.537,Z 313.52,A -85,B 0,C 180,E1 -18532.127,E2 -18532.127} C_VEL
LIN {X 0,Y 256.711,Z 313.507,A -85,B 0,C 180,E1 -18538.432,E2 -18538.432} C_VEL
LIN {X 0,Y 256.711,Z 313.502,A -85,B 0,C 180,E1 -18541.569,E2 -18541.569} C_VEL
LIN {X 0,Y 256.537,Z 313.526,A -85,B 0,C 180,E1 -18547.873,E2 -18547.873} C_VEL
LIN {X 0,Y 256.307,Z 313.558,A -85,B 0,C 180,E1 -18551.067,E2 -18551.067} C_VEL
LIN {X 0,Y 256.297,Z 313.558,A -85,B 0,C 180,E1 -18555.916,E2 -18555.916} C_VEL
LIN {X 0,Y 256.164,Z 313.57,A -85,B 0,C 180,E1 -18560.896,E2 -18560.896} C_VEL
LIN {X 0,Y 256.186,Z 313.566,A -85,B 0,C 180,E1 -18565.139,E2 -18565.139} C_VEL
LIN {X 0,Y 256.102,Z 313.578,A -85,B 0,C 180,E1 -18569.602,E2 -18569.602} C_VEL
LIN {X 0,Y 256.066,Z 313.583,A -85,B 0,C 180,E1 -18573.294,E2 -18573.294} C_VEL
LIN {X 0,Y 256.112,Z 313.58,A -85,B 0,C 180,E1 -18577.271,E2 -18577.271} C_VEL
LIN {X 0,Y 256.053,Z 313.584,A -85,B 0,C 180,E1 -18581.205,E2 -18581.205} C_VEL
LIN {X 0,Y 256.06,Z 313.777,A -85,B 0,C 180,E1 -18585.116,E2 -18585.116} C_VEL
LIN {X 0,Y 256.996,Z 316.395,A -85,B 0,C 180,E1 -18585.384,E2 -18585.384} C_VEL
LIN {X 0,Y 258.873,Z 318.845,A -85,B 0,C 180,E1 -18585.815,E2 -18585.815} C_VEL
LIN {X 0,Y 267.646,Z 333.05,A -85,B 0,C 180,E1 -18587.808,E2 -18587.808} C_VEL
LIN {X 0,Y 275.467,Z 348.379,A -85,B 0,C 180,E1 -18589.519,E2 -18589.519} C_VEL
LIN {X 0,Y 279.286,Z 357.02,A -85,B 0,C 180,E1 -18590.341,E2 -18590.341} C_VEL
LIN {X 0,Y 276.874,Z 418.321,A -85,B 0,C 180,E1 -18591.913,E2 -18591.913} C_VEL
LIN {X 0,Y 275.983,Z 431.134,A -85,B 0,C 180,E1 -18592.5,E2 -18592.5} C_VEL
LIN {X 0,Y 274.533,Z 443.832,A -85,B 0,C 180,E1 -18593.36,E2 -18593.36} C_VEL
LIN {X 0,Y 272.695,Z 454.709,A -85,B 0,C 180,E1 -18594.332,E2 -18594.332} C_VEL
LIN {X 0,Y 270.653,Z 465.89,A -85,B 0,C 180,E1 -18595.659,E2 -18595.659} C_VEL
LIN {X 0,Y 268.406,Z 476.658,A -85,B 0,C 180,E1 -18597.314,E2 -18597.314} C_VEL
LIN {X 0,Y 266.064,Z 485.601,A -85,B 0,C 180,E1 -18598.998,E2 -18598.998} C_VEL
LIN {X 0,Y 263.802,Z 493.782,A -85,B 0,C 180,E1 -18600.91,E2 -18600.91} C_VEL
LIN {X 0,Y 261.452,Z 501.755,A -85,B 0,C 180,E1 -18603.241,E2 -18603.241} C_VEL
LIN {X 0,Y 259.652,Z 507.122,A -85,B 0,C 180,E1 -18605.196,E2 -18605.196} C_VEL
LIN {X 0,Y 257.696,Z 513.108,A -85,B 0,C 180,E1 -18608.014,E2 -18608.014} C_VEL
LIN {X 0,Y 256.177,Z 517.392,A -85,B 0,C 180,E1 -18610.78,E2 -18610.78} C_VEL
LIN {X 0,Y 255.548,Z 519.247,A -85,B 0,C 180,E1 -18612.392,E2 -18612.392} C_VEL
LIN {X 0,Y 254.86,Z 521.186,A -85,B 0,C 180,E1 -18614.834,E2 -18614.834} C_VEL
LIN {X 0,Y 254.333,Z 522.16,A -85,B 0,C 180,E1 -18617.229,E2 -18617.229} C_VEL
LIN {X 0,Y 254.082,Z 522.33,A -85,B 0,C 180,E1 -18618.837,E2 -18618.837} C_VEL
LIN {X 0,Y 254.062,Z 521.411,A -85,B 0,C 180,E1 -18622.051,E2 -18622.051} C_VEL
LIN {X 0,Y 254.271,Z 519.819,A -85,B 0,C 180,E1 -18624.295,E2 -18624.295} C_VEL
LIN {X 0,Y 254.471,Z 517.021,A -85,B 0,C 180,E1 -18626.835,E2 -18626.835} C_VEL
LIN {X 0,Y 254.985,Z 513.353,A -85,B 0,C 180,E1 -18629.211,E2 -18629.211} C_VEL
LIN {X 0,Y 255.666,Z 508.585,A -85,B 0,C 180,E1 -18631.576,E2 -18631.576} C_VEL
LIN {X 0,Y 256.667,Z 502.565,A -85,B 0,C 180,E1 -18633.926,E2 -18633.926} C_VEL
LIN {X 0,Y 257.914,Z 495.092,A -85,B 0,C 180,E1 -18636.259,E2 -18636.259} C_VEL
LIN {X 0,Y 259.251,Z 487.456,A -85,B 0,C 180,E1 -18638.183,E2 -18638.183} C_VEL
LIN {X 0,Y 260.774,Z 478.166,A -85,B 0,C 180,E1 -18640.09,E2 -18640.09} C_VEL
LIN {X 0,Y 262.365,Z 467.837,A -85,B 0,C 180,E1 -18641.787,E2 -18641.787} C_VEL
LIN {X 0,Y 263.957,Z 456.367,A -85,B 0,C 180,E1 -18643.277,E2 -18643.277} C_VEL
LIN {X 0,Y 265.104,Z 444.363,A -85,B 0,C 180,E1 -18644.49,E2 -18644.49} C_VEL
LIN {X 0,Y 266.277,Z 430.941,A -85,B 0,C 180,E1 -18645.452,E2 -18645.452} C_VEL
LIN {X 0,Y 266.875,Z 418.581,A -85,B 0,C 180,E1 -18646.053,E2 -18646.053} C_VEL
LIN {X 0,Y 269.068,Z 345.39,A -85,B 0,C 180,E1 -18647.986,E2 -18647.986} C_VEL
LIN {X 0,Y 262.974,Z 328.665,A -85,B 0,C 180,E1 -18649.062,E2 -18649.062} C_VEL
LIN {X 0,Y 256.325,Z 314.286,A -85,B 0,C 180,E1 -18650.189,E2 -18650.189} C_VEL
LIN {X 0,Y 256.217,Z 313.569,A -85,B 0,C 180,E1 -18650.248,E2 -18650.248} C_VEL
LIN {X 0,Y 256.138,Z 313.568,A -85,B 0,C 180,E1 -18655.112,E2 -18655.112} C_VEL
LIN {X 0,Y 256.06,Z 313.587,A -85,B 0,C 180,E1 -18659.608,E2 -18659.608} C_VEL
LIN {X 0,Y 256.071,Z 313.589,A -85,B 0,C 180,E1 -18663.293,E2 -18663.293} C_VEL
LIN {X 0,Y 256.115,Z 313.583,A -85,B 0,C 180,E1 -18667.27,E2 -18667.27} C_VEL
LIN {X 0,Y 256.023,Z 313.587,A -85,B 0,C 180,E1 -18671.211,E2 -18671.211} C_VEL
LIN {X 0,Y 256.022,Z 313.589,A -85,B 0,C 180,E1 -18675.54,E2 -18675.54} C_VEL
LIN {X 0,Y 256.014,Z 313.586,A -85,B 0,C 180,E1 -18678.788,E2 -18678.788} C_VEL
LIN {X 0,Y 256.104,Z 313.58,A -85,B 0,C 180,E1 -18682.862,E2 -18682.862} C_VEL
LIN {X 0,Y 256.071,Z 313.578,A -85,B 0,C 180,E1 -18686.707,E2 -18686.707} C_VEL
LIN {X 0,Y 256.06,Z 313.587,A -85,B 0,C 180,E1 -18690.393,E2 -18690.393} C_VEL
LIN {X 0,Y 256.088,Z 313.571,A -85,B 0,C 180,E1 -18693.953,E2 -18693.953} C_VEL
LIN {X 0,Y 256.077,Z 313.582,A -85,B 0,C 180,E1 -18697.404,E2 -18697.404} C_VEL
LIN {X 0,Y 256.164,Z 313.573,A -85,B 0,C 180,E1 -18700.778,E2 -18700.778} C_VEL
LIN {X 0,Y 256.264,Z 313.549,A -85,B 0,C 180,E1 -18704.082,E2 -18704.082} C_VEL
LIN {X 0,Y 256.295,Z 313.556,A -85,B 0,C 180,E1 -18708.933,E2 -18708.933} C_VEL
LIN {X 0,Y 256.495,Z 313.531,A -85,B 0,C 180,E1 -18712.125,E2 -18712.125} C_VEL
LIN {X 0,Y 256.455,Z 313.53,A -85,B 0,C 180,E1 -18716.858,E2 -18716.858} C_VEL
LIN {X 0,Y 256.7,Z 313.506,A -85,B 0,C 180,E1 -18718.431,E2 -18718.431} C_VEL
LIN {X 0,Y 256.703,Z 313.507,A -85,B 0,C 180,E1 -18721.568,E2 -18721.568} C_VEL
LIN {X 0,Y 256.517,Z 313.525,A -85,B 0,C 180,E1 -18722.602,E2 -18722.602} C_VEL
LIN {X 0,Y 255.762,Z 313.621,A -85,B 0,C 180,E1 -18723.911,E2 -18723.911} C_VEL
LIN {X 0,Y 252.978,Z 313.968,A -85,B 0,C 180,E1 -18726.049,E2 -18726.049} C_VEL
LIN {X 0,Y 249.781,Z 314.366,A -85,B 0,C 180,E1 -18728.679,E2 -18728.679} C_VEL
LIN {X 0,Y 249.37,Z 314.418,A -85,B 0,C 180,E1 -18729.587,E2 -18729.587} C_VEL
LIN {X 0,Y 249.176,Z 314.446,A -85,B 0,C 180,E1 -18734.705,E2 -18734.705} C_VEL
LIN {X 0,Y 249.099,Z 314.454,A -85,B 0,C 180,E1 -18738.08,E2 -18738.08} C_VEL
LIN {X 0,Y 249.049,Z 314.461,A -85,B 0,C 180,E1 -18741.521,E2 -18741.521} C_VEL
LIN {X 0,Y 249.087,Z 314.457,A -85,B 0,C 180,E1 -18745.458,E2 -18745.458} C_VEL
LIN {X 0,Y 249.031,Z 314.468,A -85,B 0,C 180,E1 -18748.969,E2 -18748.969} C_VEL
LIN {X 0,Y 249.029,Z 314.465,A -85,B 0,C 180,E1 -18752.426,E2 -18752.426} C_VEL
LIN {X 0,Y 249.029,Z 314.465,A -85,B 0,C 180,E1 -18756.345,E2 -18756.345} C_VEL
LIN {X 0,Y 248.981,Z 314.47,A -85,B 0,C 180,E1 -18760.483,E2 -18760.483} C_VEL
LIN {X 0,Y 248.965,Z 314.473,A -85,B 0,C 180,E1 -18764.888,E2 -18764.888} C_VEL
LIN {X 0,Y 248.982,Z 314.472,A -85,B 0,C 180,E1 -18767.354,E2 -18767.354} C_VEL
LIN {X 0,Y 249.044,Z 314.464,A -85,B 0,C 180,E1 -18772.2,E2 -18772.2} C_VEL
LIN {X 0,Y 249.141,Z 314.639,A -85,B 0,C 180,E1 -18773.996,E2 -18773.996} C_VEL
LIN {X 0,Y 251.501,Z 325.319,A -85,B 0,C 180,E1 -18777.93,E2 -18777.93} C_VEL
LIN {X 0,Y 252.902,Z 332.435,A -85,B 0,C 180,E1 -18780.366,E2 -18780.366} C_VEL
LIN {X 0,Y 256.494,Z 342.701,A -85,B 0,C 180,E1 -18781.062,E2 -18781.062} C_VEL
LIN {X 0,Y 260.129,Z 371.17,A -85,B 0,C 180,E1 -18782.281,E2 -18782.281} C_VEL
LIN {X 0,Y 261.592,Z 385.822,A -85,B 0,C 180,E1 -18782.853,E2 -18782.853} C_VEL
LIN {X 0,Y 260.009,Z 441.288,A -85,B 0,C 180,E1 -18784.374,E2 -18784.374} C_VEL
LIN {X 0,Y 258.992,Z 454.576,A -85,B 0,C 180,E1 -18785.019,E2 -18785.019} C_VEL
LIN {X 0,Y 257.635,Z 467.341,A -85,B 0,C 180,E1 -18785.952,E2 -18785.952} C_VEL
LIN {X 0,Y 256.032,Z 479.473,A -85,B 0,C 180,E1 -18787.186,E2 -18787.186} C_VEL
LIN {X 0,Y 254.292,Z 491.049,A -85,B 0,C 180,E1 -18788.73,E2 -18788.73} C_VEL
LIN {X 0,Y 252.541,Z 501.474,A -85,B 0,C 180,E1 -18790.49,E2 -18790.49} C_VEL
LIN {X 0,Y 250.978,Z 511.298,A -85,B 0,C 180,E1 -18792.597,E2 -18792.597} C_VEL
LIN {X 0,Y 249.542,Z 519.915,A -85,B 0,C 180,E1 -18794.898,E2 -18794.898} C_VEL
LIN {X 0,Y 248.302,Z 527.206,A -85,B 0,C 180,E1 -18797.328,E2 -18797.328} C_VEL
LIN {X 0,Y 247.688,Z 532.132,A -85,B 0,C 180,E1 -18799.371,E2 -18799.371} C_VEL
LIN {X 0,Y 247.223,Z 536.907,A -85,B 0,C 180,E1 -18801.827,E2 -18801.827} C_VEL
LIN {X 0,Y 247.058,Z 539.467,A -85,B 0,C 180,E1 -18803.465,E2 -18803.465} C_VEL
LIN {X 0,Y 246.99,Z 541.52,A -85,B 0,C 180,E1 -18805.102,E2 -18805.102} C_VEL
LIN {X 0,Y 247.035,Z 543.151,A -85,B 0,C 180,E1 -18806.737,E2 -18806.737} C_VEL
LIN {X 0,Y 247.071,Z 544.369,A -85,B 0,C 180,E1 -18808.369,E2 -18808.369} C_VEL
LIN {X 0,Y 247.094,Z 545.143,A -85,B 0,C 180,E1 -18809.999,E2 -18809.999} C_VEL
LIN {X 0,Y 247.048,Z 545.499,A -85,B 0,C 180,E1 -18811.629,E2 -18811.629} C_VEL
LIN {X 0,Y 246.987,Z 545.464,A -85,B 0,C 180,E1 -18813.261,E2 -18813.261} C_VEL
LIN {X 0,Y 246.943,Z 544.985,A -85,B 0,C 180,E1 -18815.062,E2 -18815.062} C_VEL
LIN {X 0,Y 247.201,Z 542.96,A -85,B 0,C 180,E1 -18818.171,E2 -18818.171} C_VEL
LIN {X 0,Y 247.805,Z 540.333,A -85,B 0,C 180,E1 -18820.622,E2 -18820.622} C_VEL
LIN {X 0,Y 248.727,Z 536.711,A -85,B 0,C 180,E1 -18823.063,E2 -18823.063} C_VEL
LIN {X 0,Y 250.255,Z 532.008,A -85,B 0,C 180,E1 -18825.472,E2 -18825.472} C_VEL
LIN {X 0,Y 252.473,Z 524.957,A -85,B 0,C 180,E1 -18828.249,E2 -18828.249} C_VEL
LIN {X 0,Y 254.717,Z 517.356,A -85,B 0,C 180,E1 -18830.595,E2 -18830.595} C_VEL
LIN {X 0,Y 257.031,Z 509.607,A -85,B 0,C 180,E1 -18832.506,E2 -18832.506} C_VEL
LIN {X 0,Y 259.953,Z 499.108,A -85,B 0,C 180,E1 -18834.561,E2 -18834.561} C_VEL
LIN {X 0,Y 262.718,Z 488.446,A -85,B 0,C 180,E1 -18836.192,E2 -18836.192} C_VEL
LIN {X 0,Y 264.973,Z 478.15,A -85,B 0,C 180,E1 -18837.441,E2 -18837.441} C_VEL
LIN {X 0,Y 267.231,Z 465.858,A -85,B 0,C 180,E1 -18838.575,E2 -18838.575} C_VEL
LIN {X 0,Y 269.086,Z 452.947,A -85,B 0,C 180,E1 -18839.428,E2 -18839.428} C_VEL
LIN {X 0,Y 270.295,Z 440.506,A -85,B 0,C 180,E1 -18839.978,E2 -18839.978} C_VEL
LIN {X 0,Y 272.325,Z 387.941,A -85,B 0,C 180,E1 -18841.379,E2 -18841.379} C_VEL
LIN {X 0,Y 268.636,Z 364.069,A -85,B 0,C 180,E1 -18842.698,E2 -18842.698} C_VEL
LIN {X 0,Y 267.613,Z 359.949,A -85,B 0,C 180,E1 -18842.993,E2 -18842.993} C_VEL
LIN {X 0,Y 260.459,Z 344.318,A -85,B 0,C 180,E1 -18844.699,E2 -18844.699} C_VEL
LIN {X 0,Y 255.158,Z 334.222,A -85,B 0,C 180,E1 -18846,E2 -18846} C_VEL
LIN {X 0,Y 253.507,Z 330.667,A -85,B 0,C 180,E1 -18846.489,E2 -18846.489} C_VEL
LIN {X 0,Y 251.365,Z 322.509,A -85,B 0,C 180,E1 -18850.019,E2 -18850.019} C_VEL
LIN {X 0,Y 249.011,Z 314.469,A -85,B 0,C 180,E1 -18853.916,E2 -18853.916} C_VEL
LIN {X 0,Y 249.006,Z 314.467,A -85,B 0,C 180,E1 -18857.361,E2 -18857.361} C_VEL
LIN {X 0,Y 249.022,Z 314.459,A -85,B 0,C 180,E1 -18861.619,E2 -18861.619} C_VEL
LIN {X 0,Y 249.04,Z 314.455,A -85,B 0,C 180,E1 -18865.639,E2 -18865.639} C_VEL
LIN {X 0,Y 249.047,Z 314.457,A -85,B 0,C 180,E1 -18869.473,E2 -18869.473} C_VEL
LIN {X 0,Y 249.069,Z 314.455,A -85,B 0,C 180,E1 -18873.162,E2 -18873.162} C_VEL
LIN {X 0,Y 249.077,Z 314.452,A -85,B 0,C 180,E1 -18876.733,E2 -18876.733} C_VEL
LIN {X 0,Y 249.108,Z 314.445,A -85,B 0,C 180,E1 -18880.212,E2 -18880.212} C_VEL
LIN {X 0,Y 249.238,Z 314.429,A -85,B 0,C 180,E1 -18883.622,E2 -18883.622} C_VEL
LIN {X 0,Y 249.249,Z 314.43,A -85,B 0,C 180,E1 -18888.617,E2 -18888.617} C_VEL
LIN {X 0,Y 249.481,Z 314.399,A -85,B 0,C 180,E1 -18891.903,E2 -18891.903} C_VEL
LIN {X 0,Y 249.434,Z 314.405,A -85,B 0,C 180,E1 -18896.77,E2 -18896.77} C_VEL
LIN {X 0,Y 249.725,Z 314.37,A -85,B 0,C 180,E1 -18900,E2 -18900} C_VEL
LIN {X 0,Y 249.433,Z 314.412,A -85,B 0,C 180,E1 -18903.231,E2 -18903.231} C_VEL
LIN {X 0,Y 249.481,Z 314.405,A -85,B 0,C 180,E1 -18908.098,E2 -18908.098} C_VEL
LIN {X 0,Y 249.25,Z 314.437,A -85,B 0,C 180,E1 -18911.384,E2 -18911.384} C_VEL
LIN {X 0,Y 249.239,Z 314.436,A -85,B 0,C 180,E1 -18916.379,E2 -18916.379} C_VEL
LIN {X 0,Y 249.085,Z 314.45,A -85,B 0,C 180,E1 -18921.519,E2 -18921.519} C_VEL
LIN {X 0,Y 249.128,Z 314.445,A -85,B 0,C 180,E1 -18925.483,E2 -18925.483} C_VEL
LIN {X 0,Y 249.071,Z 314.452,A -85,B 0,C 180,E1 -18928.99,E2 -18928.99} C_VEL
LIN {X 0,Y 249.029,Z 314.456,A -85,B 0,C 180,E1 -18932.427,E2 -18932.427} C_VEL
LIN {X 0,Y 249.045,Z 314.458,A -85,B 0,C 180,E1 -18936.344,E2 -18936.344} C_VEL
